# B&R Automation Studio project JOB_NUMBER (part 4)

```iecst
END_PROGRAM

PROGRAM _EXIT
  (* Insert code here *)
END_PROGRAM
```

### Device.typ
```iecst
TYPE
	Device_typ : 	STRUCT
		RequestRelease : UINT; (*The device wants to release, Will be a line destination OR DEVICE_RELEASE_ID if not destination in bag*)
		ReadyToRecieve : BOOL; (*The device is able to recieve a bag *)
		RecieveFromID : UINT; (*(Normally 0, But when using a point with multiple options set the ID we want to release)*)
		Recieved : BOOL; (*The device has recieved a bag, instruct previous device to copy data*)
		BagInTransit : BOOL; (*The incoming device has sent a bag.*)
		ClearDestination : BOOL; (*Set this to indicate to the incoming device to clear the bag destination on data transfer.*)
		Bag : UINT; (*The bag number where to incoming device must copy data to.*)
	END_STRUCT;
END_TYPE
```

### Library Logical/http_Lib/KanHttp (IEC)
Depends on: AsHttp

#### Constants.var - Exported constants
```iecst
VAR CONSTANT
	API_UNKNOWN : USINT := 0;
	API_MAINTENANCE_CONFIRM_REENTRY : USINT := 1;
	API_CONFIG_LOAD_NEW : USINT := 2;
	API_DISCHARGER_SUBMIT : USINT := 3;
	API_DATA_ENTRY_PARTLOAD : USINT := 4;
	API_ABB_MANUAL_CMD : USINT := 10;
	API_CUSTOM_BELT_CONFIG : USINT := 90;
	API_CUSTOM_RESET_SAFETY : USINT := 91;
	API_CUSTOM_VC_COMMAND : USINT := 92;
	API_ST_FUNCTIONS : USINT := 99;
END_VAR
```

#### FindAPI.st
```iecst
(* *Get API name from URI *)
FUNCTION FindAPI

	Start := LEN(ServiceName) + 2;// We must add the / character and 1 to place the cursor on the first Letter of the API name.
	Length := FIND(URI,'?');
	IF (Length = 0) THEN
		Length := LEN(URI)- LEN(ServiceName) + 1;;
	ELSE
		Length := Length - LEN(ServiceName) - 2;
	END_IF;

	apiName := 	MID(URI,Length,Start);

	IF (apiName = 'ConfirmBagReEntry') THEN FindAPI := API_MAINTENANCE_CONFIRM_REENTRY;
	ELSIF (apiName = 'Functions') THEN FindAPI := API_ST_FUNCTIONS;
	ELSIF (apiName = 'SendBeltLoadingConfig') THEN FindAPI := API_CUSTOM_BELT_CONFIG;
	ELSIF (apiName = 'ResetSafety') THEN FindAPI := API_CUSTOM_RESET_SAFETY;
	ELSIF (apiName = 'load-config') THEN FindAPI := API_CONFIG_LOAD_NEW;
	ELSIF (apiName = 'discharger-submit') THEN FindAPI := API_DISCHARGER_SUBMIT;
	ELSIF (apiName = 'abb-manual-control') THEN FindAPI := API_ABB_MANUAL_CMD;
	ELSIF (apiName = 'part-load') THEN FindAPI := API_DATA_ENTRY_PARTLOAD;
	ELSE FindAPI := API_UNKNOWN;
	END_IF;

END_FUNCTION
```

### Program Logical/http_Lib/httpServer (IEC) - *Listen for http requests

#### _getLoadingData.st
```iecst
ACTION _getLoadingData:

	prg	:= 0;
	cat := 0;
	cus := 0;
	dst := 0;
	error := 0;
	found := 0;
	//Set common parameters of the function.
	getParameterName.searchString := requestData;
	getParameterName.searchOffset := 0;
	getParameterName.searchEndProperty := STRING_DOLLAR;

	//Find the category
	getParameterName.searchPropertyName := '"category":';
	getParameterName.searchEndProperty := ',';
	getParameterName();
	IF getParameterName.status = ERR_OK THEN
		cat := DINT_TO_UDINT(atoi(ADR(getParameterName.outputValue)));
	ELSE
		error := 2;
	END_IF;

	//Find the customer
	getParameterName.searchPropertyName := '"customer":';
	getParameterName.searchEndProperty := ',';
	getParameterName();
	IF getParameterName.status = ERR_OK THEN
		cus := DINT_TO_UDINT(atoi(ADR(getParameterName.outputValue)));
	ELSE
		error := 2;
	END_IF;

	//Find the destination
	getParameterName.searchPropertyName := '"destination":';
	getParameterName.searchEndProperty := ',';
	getParameterName();
	IF getParameterName.status = ERR_OK THEN
		dst := DINT_TO_USINT(atoi(ADR(getParameterName.outputValue)));
	ELSE
		error := 4;
	END_IF;

	//Find the program
	getParameterName.searchPropertyName := '"program":';
	getParameterName.searchEndProperty := ',';
	getParameterName();
	IF getParameterName.status = ERR_OK THEN
		prg := DINT_TO_USINT(atoi(ADR(getParameterName.outputValue)));
		bag ACCESS ADR(Bag[212]);
		found := found + 1;
		bag.Cat := cat;
		bag.Prg := prg;
		bag.Cus := cus;
		bag.Dst := dst;
	ELSE
		error := 3;
	END_IF;

	sendResponse := (found > 0);
	errorResponse := (error > 0);

END_ACTION
```

#### _httpServer.st
```iecst
ACTION _httpServer:

	//Force the server to restart when then restart the PLC. Stops the server from crashing during PLC transfer
	IF (httpServer.status = ERR_FUB_ENABLE_FALSE) THEN
		httpServer.enable := 1;
	END_IF;
	//Error Handling -- Return the code 400 (Baf if there is a process error

	IF errorResponse THEN
		responseHeader.status := '400 Bad Request';
		sendResponse := 1;
	ELSIF ton_httpTimeOut.Q THEN
		responseHeader.status := '408 Request Timeout';
		responseData := 'Response Timeout';
		sendResponse := 1;
	ELSIF sendResponse THEN;
		responseHeader.status := '200 OK';
	END_IF;

	httpServer.enable := 1;
	httpServer.send := sendResponse; // Send Response on Rising edge.
	httpServer.abort := abortResponse;	//Send abort Response on Rising Edge

	IF (overRideData.responseDataLen > 0) THEN
		httpServer.responseDataLen := overRideData.responseDataLen;
	ELSE
		httpServer.responseDataLen := brsstrlen(ADR(responseData));
	END_IF;
	IF overRideData.responseHeader.contentType <> '' THEN
		responseHeader.contentType := overRideData.responseHeader.contentType;
	ELSE
		responseHeader.contentType := 'text/plain';
	END_IF;
	IF overRideData.responseHeader.status <> '' THEN
		responseHeader.status := overRideData.responseHeader.status;
	END_IF;

	responseHeader.contentLength := httpServer.responseDataLen;

	httpServer();

	IF (httpServer.phase = httpPHASE_RECEIVED) AND NOT sendResponse THEN
		recieved := 1;
	ELSE
		recieved := 0;
	END_IF;
	//Clear the overrides
	overRideData.responseDataLen 			:= 0;
	overRideData.responseHeader				:= BLANK_RESPONSE_HEADER;

	sendResponse := 0;
	abortResponse := 0;
	errorResponse := 0;

	//Request Timeout
	ton_httpTimeOut(IN:= (httpServer.phase = httpPHASE_RECEIVED),PT:= 500);//500
END_ACTION
```

### Program Logical/http_Lib/zzHttpDriver (IEC, version 3.00.4)

#### Main.st - Init, cyclic, exit code
```iecst
//V2.00.1- First Release of Version Control - Remove all unused code- Removed temp memory for recieve data as this helps when we get a "Invalid Character error"
//V2.00.2 -- ADD: New error handling if we do not recieve data when expected.
//V2.00.3 -- ADD: Add http reply code to the http data type so we don;t have to decode the string in the user tasks
//V3.00.1 -- CHANGE: TR 23/08/2019 - Convert the driver to a state machine
//V3.00.2 -- FIX: When writing to reports the status is being set as disabled causing repeated writes -- Comment out in HTTP_CLIENT_PROCESS_REQUEST and it works.. It makes no sense!!
//V3.00.3 -- FIX: Found solution to 3.02. The original state was being set to DISABLE so the proces step was exiting incorrectly.
//V3.00.4 -- FIX: Issue with certain errors getting stuck on the abort step.
PROGRAM _INIT
	//Use Static code now but change to config file later..
	HTTP_Config.Host := '10.8.4.220';
	HTTP_Config.Port := 0;
	httpComm ACCESS ADR(HTTP_Comm[0]);

	pUrl 							:= ADR(URL);
	pRequestHeader 					:= ADR(requestHeader);
	pResponseHeader 				:= ADR(responseHeader);
	pStatistics 					:= ADR(Statistics);
	pHost 							:= ADR(requestHeader.host);

	http_Client.pUri 				:= pUrl;
	http_Client.option 				:= httpOPTION_HTTP_11;
	http_Client.pHost 				:= pHost;
	http_Client.pRequestHeader 		:= pRequestHeader;
	http_Client.pResponseHeader 	:= pResponseHeader;
	http_Client.pStatistics 		:= pStatistics;

	//Configure RequestHeader
	requestHeader.protocol := DEFAULT_REQUEST_HEADER.protocol; //'HTTP/1.1';
	requestHeader.contentType := DEFAULT_REQUEST_HEADER.contentType;//'text/plain';
	requestHeader.connection := DEFAULT_REQUEST_HEADER.connection;//'close';
	requestHeader.keepAlive := DEFAULT_REQUEST_HEADER.keepAlive;//'max=100,timeout=5';

	sizeTempMem := 500000; //Allocate 500k of free memory
	TMP_alloc(sizeTempMem,ADR(pTempMem));

	ringBuffer[0] := 0;
	//Check for any requests that were being processed on shut down..
	FOR n := 1 TO HTTP_MAX_COMM DO
		IF HTTP_Comm[n].Status = HTTP_COMM_STATUS_IN_PROCESS THEN
			ringBuffer[0] := n;
		ELSIF HTTP_Comm[n].Status = HTTP_COMM_STATUS_IN_BUFFER THEN
			ringBuffer[n] := n;
		END_IF;
	END_FOR;
	_orderRing;
END_PROGRAM

PROGRAM _CYCLIC

	//Listen to requests and add to ring buffer.
	_ringBuffer;
	http_Client.send	:= 0;
	http_Client.abort	:= 0;

	CASE httpState OF

		HTTP_CLIENT_WAIT_FOR_COMMAND: // Order the ring buffer and wait for a new command to be processed.
			http_Client.enable := 0;
			retryCount := 0;
			httpComm ACCESS ADR(HTTP_Comm[0]);
			//Wait for next command from ring buffer
			IF(ringBuffer[0] = 0) AND (ringBuffer[1] > 0) THEN
				ringBuffer[0] := ringBuffer[1];
				httpComm ACCESS ADR(HTTP_Comm[ringBuffer[0]]);
				httpComm.Status := HTTP_COMM_STATUS_IN_PROCESS;
				ringBuffer[1] := 0;
			ELSIF (ringBuffer[0] > 0) THEN
				httpState := HTTP_CLIENT_PROCESS_REQUEST;
			END_IF;

		HTTP_CLIENT_PROCESS_REQUEST:
			http_Client.enable := 0;

			replyCode := 0;
			status := HTTP_COMM_STATUS_IN_PROCESS;
			lastError := '';

			httpComm ACCESS ADR(HTTP_Comm[ringBuffer[0]]);

			brsmemcpy(ADR(URL),ADR(BLANK_CHARACTER),SIZEOF(URL));
			brsmemcpy(ADR(URL),httpComm.Command.Cmd_URL.Adr,httpComm.Command.Cmd_URL.Size);
			responseHeader := emptyResponseHeader;

			//Check for any overwrite of the host or header
			IF httpComm.Overwrite.RequestHeader THEN
				requestHeader.protocol 		:= httpComm.Overwrite.RequestHeader_Data.protocol;
				requestHeader.contentType 	:= httpComm.Overwrite.RequestHeader_Data.contentType;
				requestHeader.connection 	:= httpComm.Overwrite.RequestHeader_Data.connection;
				requestHeader.keepAlive 	:= httpComm.Overwrite.RequestHeader_Data.keepAlive;
			ELSE
				requestHeader.protocol 		:= DEFAULT_REQUEST_HEADER.protocol; //'HTTP/1.1';
				requestHeader.contentType 	:= DEFAULT_REQUEST_HEADER.contentType;//'text/plain';
				requestHeader.connection 	:= DEFAULT_REQUEST_HEADER.connection;//'close';
				requestHeader.keepAlive 	:= DEFAULT_REQUEST_HEADER.keepAlive;//'max=100,timeout=5';
			END_IF;
			IF httpComm.Overwrite.Host THEN
				requestHeader.host := httpComm.Overwrite.Host_Config.Host;
				HTTP_Config.Port := httpComm.Overwrite.Host_Config.Port;
			ELSE
				requestHeader.host := HTTP_Config.Host;
				HTTP_Config.Port := 0;
			END_IF;

			requestHeader.contentLength 	:= httpComm.Command.Body_Data.Size;
			http_Client.hostPort 			:= HTTP_Config.Port;
			http_Client.method 				:= httpComm.Command.Method;
			http_Client.pRequestData 		:= httpComm.Command.Body_Data.Adr;
			http_Client.requestDataLen 		:= httpComm.Command.Body_Data.Size;

			IF (httpComm.Command.ResponseData.Adr > 0) AND (httpComm.Command.ResponseData.Size > 0) THEN
				http_Client.pResponseData 	:= httpComm.Command.ResponseData.Adr;
				http_Client.responseDataSize := httpComm.Command.ResponseData.Size;
			ELSE
				http_Client.pResponseData := pTempMem;
				http_Client.responseDataSize := sizeTempMem;
			END_IF;
			IF (http_Client.status = ERR_FUB_ENABLE_FALSE) THEN
				httpState := HTTP_CLIENT_PROCESS_ENABLE;
			END_IF;

		HTTP_CLIENT_PROCESS_ENABLE:
			http_Client.enable := 1;
			IF (http_Client.status = ERR_OK) THEN
				httpState := HTTP_CLIENT_PROCESS_SEND;
			END_IF;

		HTTP_CLIENT_PROCESS_SEND:
			http_Client.enable := 1;
			http_Client.send := 1;
			IF (http_Client.phase = httpPHASE_SENDING) THEN
				httpState := HTTP_CLIENT_PROCESS_WAIT_RESP;
			ELSIF (http_Client.status <> ERR_OK) AND (http_Client.status <> ERR_FUB_BUSY) THEN
				httpState := HTTP_CLIENT_ABORT;
			ELSIF (http_Client.phase = httpPHASE_RECEIVED) AND (http_Client.httpStatus > 0) THEN
				httpState := HTTP_CLIENT_PROCESS_RESPONSE;
			END_IF;

		HTTP_CLIENT_PROCESS_WAIT_RESP:
			http_Client.enable := 1;
			IF (http_Client.phase = httpPHASE_RECEIVED) THEN
				httpState := HTTP_CLIENT_PROCESS_RESPONSE;
			ELSIF (http_Client.status <> ERR_OK) AND (http_Client.status <> ERR_FUB_BUSY) THEN
				httpState := HTTP_CLIENT_ABORT;
			END_IF;

		HTTP_CLIENT_PROCESS_RESPONSE:
			http_Client.enable := 1;
			IF (http_Client.status = ERR_OK) THEN
				replyCode := http_Client.httpStatus;
				CASE http_Client.httpStatus OF
					200..207:
						IF (responseHeader.contentLength > 0) THEN
							IF (responseHeader.contentLength <= httpComm.Command.ResponseData.Size) THEN
								status := HTTP_COMM_STATUS_COMPLETE;
							ELSE
								status := HTTP_COMM_STATUS_ERROR;
								lastError := 'Response data area to small';
							END_IF;
						ELSIF ((httpComm.Command.Method = httpMETHOD_POST) OR (httpComm.Command.Method = httpMETHOD_PUT)) THEN
							status := HTTP_COMM_STATUS_COMPLETE;
						END_IF;
					300..307:
						//Implementation not done
						status := HTTP_COMM_STATUS_ERROR;
						lastError := responseHeader.status;
					400..426: //Errors
						status := HTTP_COMM_STATUS_ERROR;
						lastError := responseHeader.status;
					500..510://Server Errors
						status	:= HTTP_COMM_STATUS_ERROR;
						lastError 	:= responseHeader.status;
					ELSE
						httpState 	:= HTTP_CLIENT_ABORT;
				END_CASE;
			ELSIF (http_Client.status = httpERR_BUFFER_SIZE) THEN	// Response buffer is too small -- Abort and try again with temp memory area

			ELSIF (http_Client.status <> ERR_FUB_BUSY) THEN	//http client failure.
				itoa(http_Client.status,ADR(lastError));
				httpState := HTTP_CLIENT_ABORT;
			END_IF;

			IF (status <> HTTP_COMM_STATUS_IN_PROCESS) THEN
				httpState := HTTP_CLIENT_COMPLETE;
			END_IF;

		HTTP_CLIENT_COMPLETE:
			count := count + 1;
			http_Client.enable := 0;
			httpComm.Status := status;
			httpComm.LastError := lastError;
			httpComm.ReplyCode := replyCode;
			ringBuffer[0] := 0;
			httpState := HTTP_CLIENT_WAIT_FOR_COMMAND;

		HTTP_CLIENT_ABORT:
			http_Client.enable := 1;
			http_Client.abort := 1;
			IF (http_Client.phase = httpPHASE_WAITING) OR (http_Client.phase = httpPHASE_NOT_CONNECTED)  THEN
				IF (retryCount > 0) THEN
					httpState := HTTP_CLIENT_COMPLETE;
					status := HTTP_COMM_STATUS_ERROR;
				ELSE
					retryCount := 1;
					httpState := HTTP_CLIENT_PROCESS_REQUEST;
				END_IF;
			ELSIF (http_Client.phase = httpPHASE_RECEIVED) THEN //???
				IF (retryCount > 0) THEN
					httpState := HTTP_CLIENT_COMPLETE;
					status := HTTP_COMM_STATUS_ERROR;
				ELSE
					retryCount := 1;
					httpState := HTTP_CLIENT_PROCESS_REQUEST;
				END_IF;
			END_IF;

	END_CASE;

	http_Client();

END_PROGRAM
PROGRAM _EXIT
	WHILE (http_Client.status <> ERR_OK) DO
		http_Client.enable := 1;
		http_Client.abort := 1;
		http_Client();
	END_WHILE;

END_PROGRAM
```

### Bag.typ
```iecst
TYPE
	Bag_typ : 	STRUCT
		Prg : USINT; (*Program*)
		Dst : USINT; (*Destination - Only Supertrack*)
		Wgt : UINT; (*Weight*)
		Cnt : UINT; (*Count (Items)*)
		State : UINT; (*Maintenance State WAS UR1*)
		Bid : UDINT; (*Bag ID - Supertrack ID*)
		Cat : UDINT; (*Category*)
		Mis : UDINT; (*Batch ID - MIS Mis Server*)
		Cus : UDINT; (*Customer *)
		BagNo : UDINT; (*Actual Bag Number // Was UR2*)
		Timestamp : DATE_AND_TIME;
	END_STRUCT;
END_TYPE
```

### SystemConstants.var - *SYSTEM Constants
```iecst
VAR CONSTANT
	MAX_CAMERAS : USINT := 0; (** Number of B&R Barcode scanners*)
	MAX_CONTACTRON : USINT := 0;
	MAX_DRIVES : USINT := 1; (*Set to number of drives*)
	MAX_DUAL_CHANNELS : USINT := 10; (** Number of Estops*)
	MAX_FUSE_BANKS : USINT := 0;
	MAX_HOIST : USINT := 6;
	MAX_RAILS : UINT := 201; (**DO NOT USE -> USE RAIL_COUNT INSTEAD*)
	MAX_SAFE_ZONES : USINT := 6;
END_VAR
```

### Program Logical/Standard/ABB_EPL/ABB_Driver (IEC, version 4.00.2)

#### Main.st - Init, cyclic, exit code
```iecst
//V2.00.1 -- First stable release
//V2.00.2 -- Set brake control to be optional - This means changing when we encode the paramater structure.
//V2.00.3 -- Add new constant to set MAX_FREQUENCY
//V2.00.4 -- If the drive started not on remote it wouldn;t always go into config to start. ADD new mode for when module ok is false.
//V2.00.5 -- Add test mode for simulation
//V2.00.6 -- BUG FIX -- Minumum speed was being set to Max which stopped speed control
//V2.00.7 -- REMOVE -- Remove the old structure for settings via http
//V2.00.8 -- FIX -- Correct the scaling of MaxCurrent from settings - we now us 200 = 2A
//V3.00.1 -- CHANGE Combine Settings task into driver- Remove parameters from EPL write and move to SDO configuration function block
//V3.00.2 -- ADD Manual control mode via http!
//V3.00.3 -- Convert Manual Control to mappView.
//V4.00.1 -- Automatically get node number from PV structure.
//V4.00.2 -- Move Control word states into the program as the were not being copy when the task was moved causing errors.
//V4.00.3 -- Change halt mode of belts to we do a proper decel

PROGRAM _INIT
	FOR n := 1 TO MAX_DRIVES DO
		drive ACCESS ADR(ABB_EPL.Drives[n]);
		drive.Comm.State := ABB_CONFIG;
		drive.Config.currentParam := 1; //Reset starting parameter index
		drive.Config.Node := 0;
		drive.Config.EPL_Address := '';
		index := 0;
		init_state := 0;
	END_FOR;

	FOR n := 1 TO 8 DO
		visu_manual[n].ListBoxVisible := 0;
		visu_manual[n].TargetVelocity := ABB_MIN_VELOCITY;
		visu_manual[n].selectedIndex := 0;
	END_FOR;

	IF (MAX_DRIVES > 8) THEN
		max_manualControls := 8;
	ELSIF (MAX_DRIVES > 1) THEN
		max_manualControls := MAX_DRIVES;
	ELSE
		max_manualControls := 1;
	END_IF;
	xRun := FALSE;
END_PROGRAM

PROGRAM _CYCLIC

	IF EDGENEG(xRun) THEN
		FOR n := 1 TO MAX_DRIVES DO
			drive ACCESS ADR(ABB_EPL.Drives[n]);
			drive.Comm.State := ABB_INIT;
			drive.Config.currentParam := 1; //Reset starting parameter index
			drive.Config.Node := 0;
			drive.Config.EPL_Address := '';
			index := 0;
			init_state := 0;
		END_FOR;
	ELSIF NOT xRun THEN
		_getNodeInfo;
	ELSE

		_manual;  // mappView manual control.
		FOR x := 1 TO MAX_DRIVES DO
			IF (testDrive > 0) THEN
				n := testDrive;
			ELSE
				n := x;
			END_IF;

			drive 		ACCESS ADR(ABB_EPL.Drives[n]);
			settings	ACCESS ADR(gSettings.Drive[n]);

			//Control Word												Status Word
			//Bit 0		Switch On										Bit 0	Ready To Switch On
			//Bit 1		Enable Voltage									Bit 1	Switched On
			//Bit 2		Quick Stop										Bit 2	Operation Enabled
			//Bit 3		Enable Operation								Bit 3	Fault
			//Bit 4		Not Used In Scalor Mode							Bit 4	Voltage Enabled
			//Bit 5		Not Used In Scalor Mode							Bit 5	Quick Stop
			//Bit 6		Not Used In Scalor Mode							Bit 6	Switch On Disabled
			//Bit 7		Fault Reset										Bit 7 	Warning
			//Bit 8		Halt											Bit 8	Drive Specific TBC
			//Bit 9		Operation Mode Specific							Bit 9	Remote
			//Bit 10	Reserved	??Remote Control??					Bit 10	Target Reached
			//Bit 11	Drive Specific	TBC								Bit 11 	Internal Limit Reached
			//Bit 12	Drive Specific	TBC								Bit 12	Not Used In Scalor Mode
			//Bit 13	Drive Specific	TBC								Bit 13	Not Used In Scalor Mode
			//Bit 14	Drive Specific	TBC								Bit 14	Drive Specific TBC
			//Bit 15	Drive Specific	TBC								Bit 15	Drive Specific TBC

			//Use a local instance of controlword so we don't pass changing data to the drive while processing

			controlWord := SHUT_DOWN;	// 0000 0000 0111 0110

			//Encode the controlword and statusword
			_packData;

			IF Std.TestMode AND NOT drive.Comm.ModuleOk THEN // TEST MODE
				IF drive.Cmd.Run THEN
					drive.Comm.State := ABB_RUNNING;
				ELSE
					drive.Status.ReadyToRun := 1;
				END_IF;
			ELSIF NOT drive.Comm.ModuleOk THEN
				drive.Comm.State := ABB_DISCONNECTED;
			ELSIF (drive.Config.params[MAX_PARAMS].status <> 0) OR (drive.Config.currentParam < MAX_PARAMS) THEN
				drive.Comm.State := ABB_CONFIG;
			ELSIF NOT drive.Status.OnRemote THEN
				drive.Comm.State := ABB_OFF_REMOTE;
			ELSIF drive.Status.Tripped THEN
				drive.Comm.State := ABB_TRIPPED;
			ELSIF NOT drive.Cmd.QuickStop THEN	//Enable quick stop
				drive.Comm.State := ABB_QUICK_STOP;
			ELSIF drive.Status.SwitchOnInhibit THEN
				drive.Comm.State := ABB_SWITCH_ON_INHIBITED;
			ELSIF drive.Comm.ErrorCode = ABB_FAULT_STO THEN
				drive.Comm.State := ABB_STO;
			END_IF;

			CASE drive.Comm.State OF

				ABB_DISCONNECTED:
					drive.Config.currentParam := 1; // Force write of parameters

				ABB_CONFIG: //Wait for module OK to be TRUE
					_setParameters; //Write params
					IF drive.Comm.ModuleOk AND (drive.Config.params[MAX_PARAMS].status = 0) THEN
						drive.Comm.State := ABB_SWITCH_ON_INHIBITED;
					END_IF;

				ABB_SWITCH_ON_INHIBITED:	//Wait for quick stop and enable to be true
					IF NOT drive.Status.SwitchOnInhibit THEN
						drive.Comm.State := ABB_NOT_READY_TO_SWITCH_ON;
					END_IF;

				ABB_NOT_READY_TO_SWITCH_ON:
					IF drive.Status.ReadyToSwitchOn THEN
						drive.Comm.State := ABB_READY_TO_SWITCH_ON;
					END_IF;

				ABB_READY_TO_SWITCH_ON:
					controlWord := SWITCH_ON; //0000 0111 0111
					IF drive.Status.ReadyToRun THEN
						drive.Comm.State := ABB_READY_TO_RUN;
					END_IF;

				ABB_READY_TO_RUN:
					controlWord := SWITCH_ON; //0000 0111 0111
					IF drive.Cmd.Run AND (ABS(drive.Cmd.TargetVelocity) >= ABB_MIN_VELOCITY) AND NOT drive.Manual.Enable THEN //Check min frequency is met
						drive.Comm.State := ABB_RUNNING;
					ELSIF drive.Manual.Run AND (ABS(drive.Manual.Velocity) >= ABB_MIN_VELOCITY)  THEN
						drive.Comm.State := ABB_RUNNING;
					END_IF;

				ABB_RUNNING:
					controlWord := ENABLE_OPERATION; //0000 0111 1111
					IF NOT (drive.Cmd.Run AND NOT drive.Manual.Enable) AND NOT (drive.Manual.Run AND drive.Manual.Enable) THEN
						drive.Comm.State := ABB_RAMP_DOWN;
					END_IF;

				ABB_RAMP_DOWN:
					controlWord := RAMP_DOWN; //0001 0111 1111
					IF drive.Comm.StatusWord.11 = 0 AND drive.Comm.ActVelocity = 0 THEN
						drive.Comm.State := ABB_READY_TO_RUN;
					END_IF;

				ABB_QUICK_STOP:
					controlWord := QUICK_STOP; //0000 0111 0010
					IF drive.Comm.StatusWord.11 = 0 AND drive.Comm.ActVelocity = 0 AND drive.Cmd.QuickStop THEN
						drive.Comm.State := ABB_READY_TO_RUN;
					END_IF;

				ABB_TRIPPED: // AUTO Reseting -- We should change to manual reset..
					//We must wait for the drive to be ready for reset and give an edge.
						IF (drive.Comm.StatusWord.11 = 0) AND (drive.Comm.ActVelocity = 0) THEN
							IF settings.AutoReset THEN
								controlWord := FAULT_RESET;
							ELSIF drive.Manual.ErrorReset THEN
								controlWord := FAULT_RESET;
								drive.Manual.ErrorReset := FALSE; // Reset the command.
							ELSIF (drive.Comm.ErrorCode = 0) THEN
								controlWord := FAULT_RESET; // THE FAULT HAS BEEN CLEARED EXTERNALLY
							END_IF;
						ELSE
							controlWord := DISABLE_VOLTAGE; //0000 0000 0000
						END_IF;

					//We can auto reset here..but we should log an error somewhere..
					IF NOT drive.Status.Tripped THEN
						drive.Manual.ErrorReset := FALSE; // Reset the command.
						drive.Cmd.Reset	 		:= FALSE;
						drive.Comm.State := ABB_SWITCH_ON_INHIBITED;
					END_IF;

				ABB_OFF_REMOTE:
					//Remote control not active
					controlWord := SET_REMOTE;
					////				IF drive.Status.OnRemote THEN
					////					IF (drive.Config.params[MAX_PARAMS].status <> 0) THEN
					////						drive.Comm.State := ABB_CONFIG;
					////					ELSE
					////						drive.Comm.State := ABB_SWITCH_ON_INHIBITED;
					////					END_IF;
					////				END_IF;
					//				IF NOT Std.Drives_AllowLocalMode AND (drive.Config.params[13].data = Std.Drives_AllowLocalMode) THEN //Only reset the parameters if the local control mode has chnaged
					//					_encodeParameters;
					//					drive.Config.currentParam := 1; //Reset starting parameter index
					//				END_IF;
					//
				ABB_STO:
					IF drive.Comm.ErrorCode <> ABB_FAULT_STO THEN
						drive.Comm.State := ABB_SWITCH_ON_INHIBITED;
					END_IF;

			END_CASE;
			drive.Status.Running := (drive.Comm.State =  ABB_RUNNING);
			drive.Comm.ControlWord := controlWord;

			drive.Manual := DRIVE_MANUAL_DEFAULT;
		END_FOR;

	END_IF;

	//Temp code so that we can set a node number, The NODE must already be set to 1 (DEFAULT)
	IF (newNode > 0) THEN
		setNodeNumber.enable := 1;
		setNodeNumber.node := 1;
		setNodeNumber.index := 16#4033;
		setNodeNumber.subindex := 16#03;
		setNodeNumber.pData :=  ADR(newNode);
		setNodeNumber.datalen := 2;
		setNodeNumber();
		IF (setNodeNumber.status = ERR_OK) THEN
			newNode := 0;
		END_IF;
	ELSIF saveNewNode THEN
		saveVar := 1;
		setNodeNumber.enable := 1;
		setNodeNumber.node := 1;
		setNodeNumber.index := 16#4033;
		setNodeNumber.subindex := 16#1B;
		setNodeNumber.pData :=  ADR(saveVar);
		setNodeNumber.datalen := 2;
		setNodeNumber();
		IF (setNodeNumber.status = ERR_OK) THEN
			saveNewNode := 0;
		END_IF;
	ELSIF (factoryReset > 0) THEN
		saveVar := 34560;
		setNodeNumber.enable := 1;
		setNodeNumber.node := UINT_TO_USINT(factoryReset);
		setNodeNumber.index := 16#4060;
		setNodeNumber.subindex := 16#06;
		setNodeNumber.pData :=  ADR(saveVar);
		setNodeNumber.datalen := 2;
		setNodeNumber();
		IF (setNodeNumber.status = ERR_OK) THEN
			factoryReset := 0;
		END_IF;
	END_IF;

END_PROGRAM
```

#### setParameters.st
```iecst
ACTION _setParameters:

	CASE settings.MotorSize OF // Need to set these values correctly

		ABB_MOTOR_0_25KW:
			nominalCurrent_9906		:= 7; //0.68 A
			nominalPower_9910		:= 25; // 0.37 kW
			nominalSpeed_9909 		:= 1300;
			maxCurrent				:= 190;//1.9A

		ABB_MOTOR_0_37KW_0_91A_1374:
			nominalCurrent_9906		:= 9; //0.91 A
			nominalPower_9910		:= 37; // 0.37 kW
			nominalSpeed_9909 		:= 1374;
			maxCurrent 				:= 320; //3.2A

		ABB_MOTOR_0_37KW_0_97A_1342:
			nominalCurrent_9906		:= 10; //0.97 A
			nominalPower_9910		:= 37; // 0.37 kW
			nominalSpeed_9909 		:= 1342;
			maxCurrent 				:= 350; //3.5A

		ABB_MOTOR_0_37KW_1_14A_1380:
			nominalCurrent_9906		:= 7; //1.14 A
			nominalPower_9910		:= 37; // 0.37 kW
			nominalSpeed_9909 		:= 1380;
			maxCurrent 				:= 350;//3.5A

		ABB_MOTOR_0_75KW:
			nominalCurrent_9906		:= 18; //1.75 A
			nominalPower_9910		:= 75; // 0.75 kW
			nominalSpeed_9909 		:= 1440;
			maxCurrent 				:= 1170; //11.7A

		ABB_MOTOR_1_5KW:
			nominalCurrent_9906		:= 30;// 3 A?
			nominalPower_9910		:= 150;// 1.5kW
			nominalSpeed_9909 		:= 1450;
			maxCurrent 				:= 2200; //22A ???

		ABB_MOTOR_2_2KW_4_75A_1450:
			nominalCurrent_9906		:= 48; //4.75 A
			nominalPower_9910		:= 220; // 2.2 kW
			nominalSpeed_9909 		:= 1450;
			maxCurrent 				:= 3000; //30A ???

		ABB_MOTOR_3KW:
			nominalCurrent_9906		:= 64;
			nominalPower_9910		:= 300; // 3 kW
			nominalSpeed_9909 		:= 1456;
			maxCurrent 				:= 5248; //52.48

		ABB_MOTOR_CUSTOM: // Future  Alow Motor data to be set individaully
		//			nominalCurrent_9906		:= 0;
		//			nominalPower_9910		:= 0;
		//			nominalSpeed_9909 		:= 0;
		//			maxCurrent 				:= 0;

	END_CASE;

	accTime := REAL_TO_DINT(settings.AccTime * 1000);
	decTime := REAL_TO_DINT(settings.DecTime * 1000);

	//V2.00.2 Encode parameters
	_encodeParameters;

	drive.Config.function.enable := TRUE;																	//Enable function block

	IF (drive.Config.Node > 0) THEN
		drive.Config.function.node := drive.Config.Node; 														//Node number of drive, set in ABB_EPL[n].cmd.node if non standard.
		drive.Config.function.pDevice := ADR(drive.Config.EPL_Address);											//Set powerlink address in ABB_Driver init task
	ELSE
		//drive.Config.function.node := n + 100; //Set the default to drive + 100
	END_IF;
	IF (drive.Config.Node > 0) AND (drive.Config.currentParam <= MAX_PARAMS) THEN
		IF (drive.Config.params[drive.Config.currentParam].status > 0) THEN									//Call function only if not completed
			drive.Config.function.index := drive.Config.params[drive.Config.currentParam].index; 			//Powerlink index address
			drive.Config.function.subindex := drive.Config.params[drive.Config.currentParam].subIndex;		//Powerlink sub index address
			drive.Config.function.pData := ADR(drive.Config.params[drive.Config.currentParam].data);		//Value of data to write
			drive.Config.function.datalen := drive.Config.params[drive.Config.currentParam].datalen;		//Size of data type														//Call function
			IF (drive.Config.function.status = ERR_OK) THEN 												//Clear errors
				drive.Config.params[drive.Config.currentParam].status := 0;
				drive.Config.params[drive.Config.currentParam].errorInfo := 0;
				drive.Config.currentParam := drive.Config.currentParam + 1;
			ELSIF (drive.Config.function.status <> ERR_FUB_BUSY) AND (drive.Config.function.status <> ERR_FUB_ENABLE_FALSE) THEN //Store errors
				drive.Config.params[drive.Config.currentParam].status := drive.Config.function.status;
				drive.Config.params[drive.Config.currentParam].errorInfo := drive.Config.function.errorinfo;
				drive.Config.function.enable := FALSE;
				//			ELSIF drive.Config.function.status <> 20925 THEN;//ERR_PLMGR_STATION_NOT_ACTIVE THEN  //Only skip if the devuce is active																																					//Skip if other error to stop PLC hanging in bootup
				//				drive.Config.params[drive.Config.currentParam].status := drive.Config.function.status;
				//				drive.Config.params[drive.Config.currentParam].errorInfo := drive.Config.function.errorinfo;
				//				drive.Config.currentParam := drive.Config.currentParam + 1;
			END_IF;
			drive.Config.function();
		ELSE
			drive.Config.function.enable := FALSE;
		END_IF;
	END_IF;

	//Parameters should be loaded onto default settings.
	//to default the drive set 9606 t0 34560
	//Node ID (5103) has to be manually set

END_ACTION
```

### Hoist.typ - Local data types
```iecst
TYPE
	OpcUa_type : 	STRUCT
		VC : ARRAY[100..249]OF OpcUa_VC_type;
	END_STRUCT;
	OpcUa_VC_type : 	STRUCT
		Read : OpcUa_VC_Read_type;
		Write : OpcUa_VC_Write_type;
	END_STRUCT;
	OpcUa_VC_Write_type : 	STRUCT
		Heartbeat : BOOL;
		PermissionToMove : BOOL;
		TargetPosition : USINT;
		ReleaseBag : BOOL;
		ReceiveBag : BOOL;
		LoadBag : BOOL;
		BagInTransit : BOOL;
	END_STRUCT;
	OpcUa_VC_Read_type : 	STRUCT
		StatusInfo : STRING[80];
		ActPosition : REAL;
		PositionNo : USINT;
		ReleaseBag : BOOL;
		ReceiveBag : BOOL;
		Heartbeat : BOOL;
		ReadyToReceive : BOOL;
		Auto : BOOL;
		Manual : BOOL;
		Error : BOOL;
		Weight : DINT;
		IsHome : BOOL;
		BagOnCarriage : BOOL;
		ChuteBlocked : BOOL;
	END_STRUCT;
END_TYPE
```

### Program Logical/Standard/HoistLibrary/HoistServer (IEC)

#### Variables.var
```iecst
(****************************************************)
VAR
	MTBasicsPWM_0 : MTBasicsPWM;
	i : USINT;
	pHmiOpcUa : REFERENCE TO OpcUa_VC_type;
	selectedVC : UINT;
	pulse : MTBasicsPWM;
	hoist : REFERENCE TO OpcUa_VC_type;
	ton_simulateRecv : ARRAY[230..249] OF TON;
END_VAR
```

#### Main.st
```iecst
//V1.00.1  - TR - Add simulution mode.

PROGRAM _INIT

	selectedVC := 240;

END_PROGRAM

PROGRAM _CYCLIC

	MTBasicsPWM_0.DutyCycle		:= 50;
	MTBasicsPWM_0.Period		:= 2;
	MTBasicsPWM_0.Enable		:= TRUE;
	MTBasicsPWM_0(Enable:= TRUE,DutyCycle:= 50,Period:= 2,Update := 1);

	//FOR i := 38 TO 39 DO

pHmiOpcUa ACCESS ADR(OpcUa.VC[selectedVC]);

IF Std.TestMode THEN
		FOR i := 231 TO 249 DO

			hoist ACCESS ADR (OpcUa.VC[i]);

			hoist.Read.PositionNo 			:=	hoist.Write.TargetPosition;
			hoist.Read.Auto							:= 1;
			hoist.Read.ReadyToReceive 	:= 1;
			hoist.Read.IsHome						:= 1;

			ton_simulateRecv[i].IN 			:= 	hoist.Write.ReceiveBag;
			ton_simulateRecv[i].PT 			:= T#5s;
			ton_simulateRecv[i]();

			hoist.Read.ReceiveBag := ton_simulateRecv[i].Q;

			IF ton_simulateRecv[i].Q THEN
				hoist.Read.BagOnCarriage := 1;
			ELSIF hoist.Write.ReleaseBag THEN
				hoist.Read.BagOnCarriage := 0;
			END_IF;

		END_FOR;

ELSE
		FOR i := 231 TO 249 DO
			OpcUa.VC[i].Write.Heartbeat	:= MTBasicsPWM_0.Out; // NOT OpcUa.VC[i].Write.Heartbeat;
			//OpcUa.VC[i].Write.Heartbeat	:= pulse.Out;

			OpcUa.VC[i].Read.StatusInfo;
			OpcUa.VC[i].Read.ActPosition;
			OpcUa.VC[i].Read.PositionNo;
			OpcUa.VC[i].Read.ReceiveBag;
			OpcUa.VC[i].Read.ReleaseBag;
			OpcUa.VC[i].Read.Heartbeat;
			OpcUa.VC[i].Read.ReadyToReceive;

		END_FOR;

END_IF;

	(* Establish a connection to the client *)

(*	ReadHeartbeat;

	CASE Connect_to_OpcUaServer_step OF

		WAIT:

			IF Connect_OpcUa THEN

				Connect_to_OpcUaServer_step := CONNECT_TO_OPCUA;
			END_IF;

		CONNECT_TO_OPCUA:

			SessionConnectInfo_0.SecurityMsgMode := UASecurityMsgMode_None;
			SessionConnectInfo_0.SecurityPolicy := UASecurityPolicy_None;
			SessionConnectInfo_0.TransportProfile := UATP_UATcp;
			SessionConnectInfo_0.UserIdentityToken.UserIdentityTokenType := UAUITT_Anonymous;
			SessionConnectInfo_0.SessionTimeout := T#10m;
			SessionConnectInfo_0.MonitorConnection := T#10s;

			UA_Connect_0.ServerEndpointUrl := 'opc.tcp://10.44.10.244:4840';
			UA_Connect_0.Timeout := T#10s;
			UA_Connect_0.Execute := TRUE;
			UA_Connect_0.SessionConnectInfo := SessionConnectInfo_0;

			IF (UA_Connect_0.Done = 1) THEN
				UA_Connect_0.Execute := FALSE;
				Connect_OpcUa := FALSE;
				ConnectionHdl := UA_Connect_0.ConnectionHdl;
				Connect_to_OpcUaServer_step := GET_NAMESPACE;
			END_IF;

			IF (UA_Connect_0.Error = 1) THEN
				ConnectionHdl := 0;
				UA_Connect_0.Execute := FALSE;
				Connect_to_OpcUaServer_step := ERROR_OPCUA;
			END_IF;

		GET_NAMESPACE:

			UA_GetNamespaceIndex_0.ConnectionHdl := ConnectionHdl;
			UA_GetNamespaceIndex_0.NamespaceUri := 'urn:B&R/pv/';
			UA_GetNamespaceIndex_0.Timeout := T#5s;
			UA_GetNamespaceIndex_0.Execute := TRUE;

			IF (UA_GetNamespaceIndex_0.Done = 1) THEN
				NamespaceIndex := UA_GetNamespaceIndex_0.NamespaceIndex;
				UA_GetNamespaceIndex_0.Execute := FALSE;
				Connect_to_OpcUaServer_step := GET_NODE_HANDLE;
			END_IF;

			IF (UA_GetNamespaceIndex_0.Error = 1) THEN
				NamespaceIndex := 0;
				UA_GetNamespaceIndex_0.Execute := FALSE;
				Connect_to_OpcUaServer_step := ERROR_OPCUA;
			END_IF;

		GET_NODE_HANDLE:

			UANodeID_0[0].NamespaceIndex := NamespaceIndex;
			UANodeID_0[0].Identifier := '::Test_OpcUa_Client:WriteHeartbeat';
			UANodeID_0[0].IdentifierType := UAIdentifierType_String;

			UA_NodeGetHandleList_0.ConnectionHdl := ConnectionHdl;
			UA_NodeGetHandleList_0.NodeIDCount := 1;
			UA_NodeGetHandleList_0.NodeIDs := UANodeID_0;
			UA_NodeGetHandleList_0.Timeout := T#10s;
			UA_NodeGetHandleList_0.Execute := TRUE;

			IF (UA_NodeGetHandleList_0.Done = 1) THEN
				NodeHdls := UA_NodeGetHandleList_0.NodeHdls;
				UA_NodeGetHandleList_0.Execute := FALSE;
				Connect_to_OpcUaServer_step := READ_LIST;
			END_IF;

			IF (UA_NodeGetHandleList_0.Error = 1) THEN
				NodeHdls[0] := 0;

				UA_NodeGetHandleList_0.Execute := FALSE;
				Connect_to_OpcUaServer_step := ERROR_OPCUA;
			END_IF;

		READ_LIST:

			UANodeAdditionalInfo_0[0].AttributeId := UAAI_Value;
			UANodeAdditionalInfo_0[0].IndexRangeCount := 0;

			Variable_Rd0[0] := '::ServerTask:ReadHeartbeat';

			IF NOT UA_ReadList_0.Done THEN

				UA_ReadList_0
					(
					Execute := TRUE,
					ConnectionHdl := ConnectionHdl,
					NodeHdlCount := 1,
					NodeHdls := NodeHdls,
					NodeAddInfo := UANodeAdditionalInfo_0,
					Timeout := T#10s,
				Variables := Variable_Rd0);

				IF (UA_ReadList_0.Busy = 0) THEN
					UA_ReadList_0.Execute := FALSE;

					IF (UA_ReadList_0.Done = 1) THEN
						TimestampHeart := UA_ReadList_0.TimeStamps[0];

					END_IF;
					IF (UA_ReadList_0.Error = 1) THEN
						TimestampHeart := 0;
						Connect_to_OpcUaServer_step := ERROR_OPCUA;
					END_IF;
				END_IF;

			ELSIF StopReading THEN
				Connect_to_OpcUaServer_step := RELEASE_NODE;
				UA_ReadList_0.Execute := FALSE;

			ELSE
				UA_ReadList_0
					(
					Execute := FALSE,
					ConnectionHdl := ConnectionHdl,
					NodeHdlCount := 1,
					NodeHdls := NodeHdls,
					NodeAddInfo := UANodeAdditionalInfo_0,
					Timeout := T#10s,
				Variables := Variable_Rd0);
			END_IF;

		RELEASE_NODE:

			UA_NodeReleaseHandleList_0.ConnectionHdl := ConnectionHdl;
			UA_NodeReleaseHandleList_0.NodeHdlCount := 1;
			UA_NodeReleaseHandleList_0.NodeHdls := NodeHdls;
			UA_NodeReleaseHandleList_0.Timeout := T#10s;
			UA_NodeReleaseHandleList_0.Execute := TRUE;
			StopReading := FALSE;

			IF (UA_NodeReleaseHandleList_0.Done = 1) THEN
				NodeHdls[0] := 0;

				UA_NodeReleaseHandleList_0.Execute := FALSE;
				Connect_to_OpcUaServer_step := DISCONNECT_OPCUA;
			END_IF;

			IF (UA_NodeReleaseHandleList_0.Error = 1) THEN
				NodeHdls[0] := 0;

				UA_NodeReleaseHandleList_0.Execute := FALSE;
				Connect_to_OpcUaServer_step := ERROR_OPCUA;
			END_IF;

		DISCONNECT_OPCUA:

			UA_Disconnect_0.ConnectionHdl := ConnectionHdl;
			UA_Disconnect_0.Timeout := T#10s;
			UA_Disconnect_0.Execute := TRUE;

			IF (UA_Disconnect_0.Done = 1) THEN
				ConnectionHdl := 0;
				UA_Disconnect_0.Execute := FALSE;
				Connect_to_OpcUaServer_step := WAIT;
			END_IF;

			IF (UA_Disconnect_0.Error = 1) THEN
				ConnectionHdl := 0;
				UA_Disconnect_0.Execute := FALSE;
				Connect_to_OpcUaServer_step := ERROR_OPCUA;
			END_IF;

		ERROR_OPCUA:

	END_CASE;

	UA_Connect_0;
	UA_GetNamespaceIndex_0;
	UA_NodeGetHandleList_0;
	UA_NodeReleaseHandleList_0;
	UA_Disconnect_0;				*)

END_PROGRAM

PROGRAM _EXIT
	(* Insert code here *)

END_PROGRAM
```

### IOlink.typ
```iecst
TYPE
	contactron_visu_manual_typ : 	STRUCT
		Visible : BOOL; (**Are the controls Visible*)
		Name : STRING[50];
		Address : STRING[80]; (*Reference to the phyical location*)
		CommOk : BOOL;
		ActCurrent : DINT;
		ErrorCode : UINT;
		RunReverse : BOOL;
		RunForwards : BOOL;
		SetCurrent : INT;
		ErrorReset : BOOL;
		ErrorActive : BOOL;
		selectedIndex : UINT;
		selectedValue : STRING[10];
		refreshDropDown : R_TRIG;
		ListBoxVisible : BOOL;
		EnableRunReverse : BOOL;
		EnableRunForwards : BOOL;
		Enable : BOOL;
		Node : USINT;
	END_STRUCT;
	Contactron_Cmd_Type : 	STRUCT
		Reset_Manual : BOOL;
		Reset_Automatic : BOOL;
		Stop : BOOL;
		Run : BOOL;
		Direction : Contactron_Direction;
		Current : USINT; (*Sets the trip current, enable must be off to write*)
	END_STRUCT;
	Contactron_Comms_Type : 	STRUCT
		Write : Contactron_Outputs_Type;
		Read : Contactron_Inputs_Type;
	END_STRUCT;
	Contactron_Device_Type :
		(
		CONTACTRON_H5_3 := 0,
		CONTACTRON_H5_9 := 1,
		CONTACTRON_H3_3 := 2,
		CONTACTRON_H3_9 := 3
		);
	Contactron_Direction :
		(
		CONTACTRON_FORWARD := 0,
		CONTACTRON_REVERSE := 1
		);
	Contactron_Inputs_Type : 	STRUCT
		Diagnostics : USINT;
		CurrentStatus : USINT; (*Current trip level and trip status*)
		ThermalPercentOfMax : USINT;
		CurrentPercentOfMax : USINT;
		DeviceType : USINT; (*Type of contactron used*)
		CurrentActual : USINT; (*10mA*)
		Data : ARRAY[0..5]OF USINT;
	END_STRUCT;
	Contactron_Outputs_Type : 	STRUCT
		Control : USINT;
		NominalCurrent : USINT;
	END_STRUCT;
	Contactron_Status_Type : 	STRUCT
		Error : BOOL;
		STO_Active : BOOL;
		Device_Ok : BOOL;
		Overload_Warning : BOOL;
		MainsFailure : BOOL;
		PhaseLoss : BOOL;
		Current : REAL;
		DeviceType : Contactron_Device_Type;
	END_STRUCT;
	Contactron_Type : 	STRUCT  (*Parent structure to hold all Contactron structures*)
		Cmd : Contactron_Cmd_Type;
		Status : Contactron_Status_Type;
		Comms : Contactron_Comms_Type;
		Manual : contactron_visu_manual_typ;
	END_STRUCT;
	IO_Link_Type : 	STRUCT  (*Parent structure to hold all IO_Link device structures*)
		Contactron : ARRAY[0..MAX_CONTACTRON]OF Contactron_Type; (*Parent structure to hold all Contactron structures*)
	END_STRUCT;
END_TYPE

(**)
```

### Program Logical/Standard/IOLink/Contactron/Contactron (IEC, version 1.00.2)

#### Main.st - Init, cyclic, exit code
```iecst
(********************************************************************
 * COPYRIGHT --
 ********************************************************************
 * PROGRAM: IOLink
 * File: IOLink_Driver.s
 * Author: Stephen Healy NOT ANYMORE :)
 * Created: Sept 05, 2018
 ********************************************************************
 * Implementation OF PROGRAM IOLink
 ********************************************************************)
//V1.00.1 First Release
//V1.00.1 TR 10/11/2020  - Remove run signal from contactron when there is a fault to allow the error to be acknowledged.
//V1.00.2 TR 07/04/2021  - Add Test mode

PROGRAM _INIT

END_PROGRAM

PROGRAM _CYCLIC

	//Call contactron action
	IF MAX_CONTACTRON > 0 THEN
		_visu;
		_Contactron;

	END_IF;

END_PROGRAM
```

#### Variables.var - Local variables
```iecst
VAR
	n : UINT;
END_VAR
VAR CONSTANT
	max_manualControls : USINT := 8;
END_VAR
VAR
	visu_man : REFERENCE TO contactron_visu_manual_typ;
	visu_manual : ARRAY[0..max_manualControls] OF contactron_visu_manual_typ;
	selIndex : DINT;
	updateDropDown : BOOL;
	index : UINT;
	manualSelectDrowDown : ARRAY[0..MAX_CONTACTRON] OF STRING[125];
	sIndex : STRING[10];
	run : BOOL;
	contactron : REFERENCE TO Contactron_Type;
	RunMotor : BOOL;
	name : STRING[30];
END_VAR
VAR CONSTANT
	CONTACTRON_MANUAL_DEFAULT : contactron_visu_manual_typ := (RunReverse:=FALSE,RunForwards:=FALSE,ErrorReset:=FALSE,Enable:=FALSE);
END_VAR
```

#### _Contactron.st
```iecst
ACTION _Contactron:
	//----------------------------------------------
	//-----------------Contactron-------------------
	//----------------------------------------------

	//Write control word
	FOR n:=1 TO MAX_CONTACTRON DO
		contactron ACCESS ADR(IO_Link.Contactron[n]);

		IF Std.TestMode  THEN
			contactron.Status.Device_Ok := 1;
			IF contactron.Cmd.Run THEN
				contactron.Status.Current := 1.0;
			ELSE
				contactron.Status.Current := 0.0;
			END_IF;

		ELSE
			contactron.Comms.Read.CurrentActual 		:= contactron.Comms.Read.Data[0];
			contactron.Comms.Read.DeviceType 			:= contactron.Comms.Read.Data[1];
			contactron.Comms.Read.ThermalPercentOfMax 	:= contactron.Comms.Read.Data[2];
			contactron.Comms.Read.CurrentPercentOfMax 	:= contactron.Comms.Read.Data[3];
			contactron.Comms.Read.CurrentStatus 		:= contactron.Comms.Read.Data[4];
			contactron.Comms.Read.Diagnostics 			:= contactron.Comms.Read.Data[5];

			//Read status
			contactron.Status.Error 			:= contactron.Comms.Read.Diagnostics.0;
			contactron.Status.STO_Active 		:= NOT contactron.Comms.Read.Diagnostics.3;
			contactron.Status.Device_Ok 		:= contactron.Comms.Read.Diagnostics.5;
			contactron.Status.Overload_Warning 	:= contactron.Comms.Read.Diagnostics.6;
			contactron.Status.MainsFailure 		:= ((contactron.Comms.Read.CurrentStatus AND CONTACTRON_TRIP_STATUS) = CONTACTRON_MAINS_LOSS);
			contactron.Status.PhaseLoss 		:= ((contactron.Comms.Read.CurrentStatus AND CONTACTRON_TRIP_STATUS) = CONTACTRON_PHASE_LOSS);
			contactron.Status.Current 			:= contactron.Comms.Read.CurrentActual * 0.01;
			contactron.Status.DeviceType 		:= contactron.Comms.Read.DeviceType;

			IF contactron.Status.Error THEN
				run := 0;
//			ELSE IF contactron.Manaual.enable THEN
//				run := Manaul.run.
			ELSE
				run := contactron.Cmd.Run;
			END_IF;

			CASE contactron.Cmd.Direction OF
				CONTACTRON_FORWARD:
					contactron.Comms.Write.Control.0 := run;
					contactron.Comms.Write.Control.7 := run;
					contactron.Comms.Write.Control.1 := FALSE;
					contactron.Comms.Write.Control.5 := FALSE;

				CONTACTRON_REVERSE:
					contactron.Comms.Write.Control.0 := FALSE;
					contactron.Comms.Write.Control.7 := FALSE;
					contactron.Comms.Write.Control.1 := run;
					contactron.Comms.Write.Control.5 := run;

				ELSE
					contactron.Comms.Write.Control.0 := FALSE;
					contactron.Comms.Write.Control.7 := FALSE;
					contactron.Comms.Write.Control.1 := FALSE;
					contactron.Comms.Write.Control.5 := FALSE;

			END_CASE;

			contactron.Comms.Write.Control.2 := contactron.Cmd.Reset_Manual;
			contactron.Comms.Write.Control.3 := contactron.Cmd.Reset_Automatic;
			contactron.Comms.Write.Control.4 := FALSE; //NOT USED
			contactron.Comms.Write.Control.6 := contactron.Cmd.Stop;

			IF contactron.Cmd.Current > 0 THEN //Write trip current level
				contactron.Comms.Write.NominalCurrent := (contactron.Cmd.Current OR CONTACTRON_WRITE_CURRENT);
			ELSE
				contactron.Comms.Write.NominalCurrent := 0;
			END_IF;
			IF contactron.Cmd.Current = (contactron.Comms.Read.CurrentStatus AND CONTACTRON_CURRENT_STATUS) THEN
				contactron.Cmd.Current := 0; //Reset trip current if cmd written
			END_IF;

		END_IF;

		//Clear the manual commands.
		contactron.Manual := CONTACTRON_MANUAL_DEFAULT;
	END_FOR;
END_ACTION
```

#### _visu.st
```iecst
ACTION _visu:

	FOR n := 1 TO max_manualControls DO

		visu_man ACCESS ADR(visu_manual[n]);

		selIndex := atoi(ADR(visu_man.selectedValue));
		IF (selIndex > 0) AND (selIndex <= MAX_CONTACTRON) AND (selIndex <> visu_man.selectedIndex) THEN
			updateDropDown := 1;
			visu_man.selectedIndex := DINT_TO_UINT(selIndex);
		END_IF;

		visu_man.ListBoxVisible := (visu_man.selectedIndex = 0);

		visu_man.refreshDropDown.CLK := (visu_man.selectedIndex = 0);
		visu_man.refreshDropDown();
		IF visu_man.refreshDropDown.Q THEN
			updateDropDown := 1;
		END_IF;

		contactron ACCESS ADR(IO_Link.Contactron[visu_man.selectedIndex]);
		contactron.Manual.Enable := 1; //Mark Contactron as in manual mode

		visu_man.Visible 		:= (visu_man.selectedIndex >0);
		visu_man.Name    		:= gSettings.Contactron[visu_man.selectedIndex].Name;
//		visu_man.Node	 		:=
		visu_man.CommOk  		:= contactron.Status.Device_Ok;
		visu_man.ActCurrent 	:= contactron.Comms.Read.CurrentActual;
		visu_man.ErrorCode 		:= contactron.Status.Error;

		visu_man.ErrorActive := (contactron.Status.Error);

//		drive ACCESS ADR(ABB_EPL.Drives[visu_man.selectedIndex]);
//		drive.Manual.Enable 	:= 1; // Mark the drive as in manual mode.
//		drive.Manual.Velocity 	:= visu_man.TargetVelocity;
//
//		visu_man.Visible		:= (visu_man.selectedIndex > 0);
//		visu_man.Name			:= gSettings.Drive[visu_man.selectedIndex].Name;
//		visu_man.Node		 	:= drive.Config.Node;
//		visu_man.ModuleOk 		:= drive.Comm.ModuleOk;
//		visu_man.ActVelocity 	:= ABS(drive.Comm.ActVelocity);
//		visu_man.ActCurrent 	:= drive.Comm.ActCurrent;
//		visu_man.ActTorque 		:= drive.Comm.ActTorque;
//		visu_man.ErrorCode 		:= drive.Comm.ErrorCode;
//
//		visu_man.ErrorActive	:= (drive.Comm.State = ABB_TRIPPED);
//
		IF visu_man.ErrorReset THEN
			visu_man.ErrorReset := 0;
			contactron.Manual.ErrorReset := 1;
		END_IF;

//		CASE drive.Comm.State OF
//			ABB_INIT:
//				visu_man.State := '$$Drives.State.Init';
//			ABB_DISCONNECTED:
//				visu_man.State := '$$Drives.State.Disconnected';
//			ABB_QUICK_STOP:
//				visu_man.State := '$$Drives.State.QuickStop';
//			ABB_CONFIG:
//				visu_man.State := '$$Drives.State.Config';
//			ABB_SWITCH_ON_INHIBITED:
//				visu_man.State := '$$Drives.State.SwitchOnInhibit';
//			ABB_NOT_READY_TO_SWITCH_ON:
//				visu_man.State := '$$Drives.State.NotReady';
//			ABB_READY_TO_SWITCH_ON:
//				visu_man.State := '$$Drives.State.ReadyToSwitchOn';
//			ABB_READY_TO_RUN:
//				visu_man.State := '$$Drives.State.ReadyToRun';
//			ABB_RUNNING:
//				visu_man.State := '$$Drives.State.Running';
//			ABB_TRIPPED:
//				visu_man.State := '$$Drives.State.Tripped';
//			ABB_OFF_REMOTE:
//				visu_man.State := '$$Drives.State.OffRemote';
//			ABB_STO:
//				visu_man.State := '$$Drives.State.STO';
//			ABB_RAMP_DOWN:
//				visu_man.State := '$$Drives.State.RampDown';
//			ELSE
//				visu_man.State := '';
//		END_CASE;
//
		RunMotor := (contactron.Status.Device_Ok) AND NOT (contactron.Status.Error);
//		targetSpeedValid := ((visu_man.TargetVelocity >= ABB_MIN_VELOCITY) AND (visu_man.TargetVelocity <= ABB_MAX_VELOCITY) AND ((drive.Comm.State = ABB_READY_TO_RUN) OR  (drive.Comm.State = ABB_RUNNING)));
		//
		IF NOT visu_man.Enable THEN
			visu_man.RunReverse				:= 0;
			visu_man.RunForwards			:= 0;
			visu_man.EnableRunReverse   	:= 0;
			visu_man.EnableRunForwards		:= 0;
		ELSIF visu_man.RunForwards THEN
			contactron.Manual.RunForwards 	:= 1;
			contactron.Cmd.Run				:= RunMotor;
			visu_man.EnableRunReverse	  	:= 0;
		ELSIF visu_man.RunReverse THEN
			contactron.Manual.RunReverse	:= 1;
			contactron.Cmd.Run				:= RunMotor;
			visu_man.EnableRunForwards		:= 0;
		ELSE
			visu_man.EnableRunReverse		:= 1;
			visu_man.EnableRunForwards		:= 1;
		END_IF;

//		IF NOT targetSpeedValid THEN
//			visu_man.RunReverse 		:= 0;
//			visu_man.RunForwards 		:= 0;
//			visu_man.EnableRunReverse 	:= 0;
//			visu_man.EnableRunForwards 	:= 0;
//		ELSIF visu_man.RunForwards THEN
//			drive.Manual.Direction 	:= ABB_DIRECTION_FWD;
//			drive.Manual.Run		:= targetSpeedValid;
//			visu_man.EnableRunReverse := 0;
//		ELSIF visu_man.RunReverse THEN
//			drive.Manual.Direction 	:= ABB_DIRECTION_REV;
//			drive.Manual.Run		:= targetSpeedValid;
//			visu_man.EnableRunForwards := 0;
//		ELSE
//			visu_man.EnableRunReverse := 1;
//			visu_man.EnableRunForwards := 1;
//			drive.Manual.Run		:= 0;
//		END_IF;

	END_FOR;

	//Build the list box string;
	//[{'value':'text_1', 'text':'$$IAT/testText1'}, {'value':'text_2', 'text':'$$IAT/testText2'}]
	IF updateDropDown THEN
		index := 1;
		brsmemset(ADR(manualSelectDrowDown),0,SIZEOF(manualSelectDrowDown));
		manualSelectDrowDown[0] := '{"value":0,"text":""}';
		FOR n := 1 TO MAX_CONTACTRON DO
			contactron ACCESS ADR(IO_Link.Contactron[n]);
			IF NOT contactron.Manual.Enable THEN
				itoa(n,ADR(sIndex));

				IF (gSettings.Contactron[n].Name <> '') THEN
					name := gSettings.Contactron[n].Name;
				ELSE
					name := 'C ';
					brsstrcat(ADR(name),ADR(sIndex));
				END_IF;
				brsstrcat(ADR(manualSelectDrowDown[index]),ADR('{"value":"'));
				brsstrcat(ADR(manualSelectDrowDown[index]),ADR(sIndex));
				brsstrcat(ADR(manualSelectDrowDown[index]),ADR('","text":"'));
				brsstrcat(ADR(manualSelectDrowDown[index]),ADR(name));
				brsstrcat(ADR(manualSelectDrowDown[index]),ADR('"}'));
				index := index + 1;
			END_IF;
		END_FOR;
		updateDropDown := FALSE;
	END_IF;

END_ACTION
```

### Program Logical/Standard/IOLink/FuseManagement (IEC, version 1.00.2)

#### Main.st - Init, cyclic, exit code
```iecst
//V1.00.0 -- First Release
//V1.00.1 -- Update so we monitor the status of the fuse and can send reset commands
//V1.00.2 -- Invert the fault lamp to a healthy lamp to stay consistent with hardwired devices

PROGRAM _INIT
Fuse[1].pDevice := ADR('SL1.IF1.ST11.IF1.ST9.IF1');//'SL1.IF1.ST2.IF1.ST7.IF1');
Fuse[2].pDevice := ADR('SL1.IF1.ST11.IF1.ST9.IF2');
Fuse[3].pDevice := ADR('SL1.IF1.ST11.IF1.ST9.IF3');
Fuse[4].pDevice := ADR('SL1.IF1.ST11.IF1.ST9.IF4');
Fuse[5].pDevice := ADR('SL1.IF1.ST11.IF1.ST10.IF1');
Fuse[6].pDevice := ADR('SL1.IF1.ST11.IF1.ST10.IF2');
Fuse[7].pDevice := ADR('SL1.IF1.ST21.IF1.ST9.IF1');
Fuse[8].pDevice := ADR('SL1.IF1.ST21.IF1.ST9.IF2');
Fuse[9].pDevice := ADR('SL1.IF1.ST21.IF1.ST9.IF3');
Fuse[10].pDevice := ADR('SL1.IF1.ST21.IF1.ST9.IF4');
Fuse[11].pDevice := ADR('SL1.IF1.ST21.IF1.ST10.IF1');
Fuse[12].pDevice := ADR('SL1.IF1.ST21.IF1.ST10.IF2');
Fuse[13].pDevice := ADR('SL1.IF1.ST61.IF1.ST5.IF3');
Fuse[14].pDevice := ADR('SL1.IF1.ST61.IF1.ST5.IF4');
Fuse[15].pDevice := ADR('SL1.IF1.ST62.IF1.ST5.IF3');
Fuse[16].pDevice := ADR('SL1.IF1.ST62.IF1.ST5.IF4');
Fuse[17].pDevice := ADR('SL1.IF1.ST63.IF1.ST5.IF3');
Fuse[18].pDevice := ADR('SL1.IF1.ST63.IF1.ST5.IF4');

FOR n := 1 TO MAX_FUSE_BANKS DO
	fuse ACCESS ADR(Fuse[n]);
	fuse.Write.MinVoltage := 1500;
	fuse.Write.MaxVoltage := 2800;
	FOR i := 1 TO MAX_FUSES DO
      fuse.Write.Channel[i].Status := EB_STATE_ON;
      fuse.Write.Channel[i].TripCurrent := 40;
  END_FOR;
	fuse.index := 90;
	fuse.readStatusOnly := 0;
	fuseTrippedAlarm[n] := 0;
END_FOR;

//alarm 	ACCESS ADR(Alarm[208]);
END_PROGRAM

PROGRAM _CYCLIC

IF EDGEPOS(X[1003].X04) THEN
	reset[0] := 1;
END_IF;
IF EDGEPOS(X[2003].X04) THEN
	reset[1] := 1;
END_IF;

fuseFault[0] := 0;
fuseFault[1] := 0;
//alarm.On	:= 0;
//alarm.Name	:= 0;

FOR n := 1 TO MAX_FUSE_BANKS DO
	fuse ACCESS ADR(Fuse[n]);
	read ACCESS ADR(fuse.IOLinkRead);
	write ACCESS ADR(fuse.IOLinkWrite);

	read.enable := 1;
	write.enable := 1;
	write.pDeviceName 	:= fuse.pDevice;
	read.pDeviceName 	:= fuse.pDevice;

	IF EDGEPOS(read.readLen > 0) THEN
		count := count + 1;
	END_IF;

	IF (read.errorCode > 0) THEN
		fuse.index := 10;
	END_IF;

	IF (n < 5) THEN
		plc := 0;
	ELSE
		plc := 1;
	END_IF;

	CASE fuse.index	OF
		0:

		32:	//Read Error Count
			read.datatype 		:= ioLinkTYPE_SINT;
			read.pData			:= ADR(fuse.Read.ErrorCount);
			read.dataLen		:= SIZEOF(fuse.Read.ErrorCount);
			read.index			:= fuse.index;
			read.subIndex		:= 0;
			read();
			IF read.status = ERR_OK THEN
				fuse.index := fuse.index + 1;
			ELSIF (read.status <> ERR_FUB_BUSY) AND (read.status <> ERR_FUB_ENABLE_FALSE)  THEN
				fuse.index := fuse.index + 1;
				//fuse.Read.ErrorCount := 0;
			END_IF;

		33://
			fuse.index := 36;

		36://Device Status	 R/O USINT
			read.datatype 		:= ioLinkTYPE_SINT;
			read.pData			:= ADR(fuse.Read.DeviceStatus);
			read.dataLen		:= SIZEOF(fuse.Read.DeviceStatus);
			read.index			:= fuse.index;
			read.subIndex		:= 0;
			read();
			IF read.status = ERR_OK THEN
				fuse.index := fuse.index + 1;
			ELSIF (read.status <> ERR_FUB_BUSY) AND (read.status <> ERR_FUB_ENABLE_FALSE)  THEN
				fuse.index := fuse.index + 1;
				//fuse.Read.ErrorCount := 0;
			END_IF;

		37:// Device Status	 R/O String
			read.datatype 		:= ioLinkTYPE_STRING;
			read.pData			:= ADR(fuse.Read.DeviceStatusString);
			read.dataLen		:= SIZEOF(fuse.Read.DeviceStatusString);
			read.index			:= fuse.index;
			read.subIndex		:= 0;
			read();
			IF read.status = ERR_OK THEN
				fuse.index := fuse.index + 1;
			ELSIF (read.status <> ERR_FUB_BUSY) AND (read.status <> ERR_FUB_ENABLE_FALSE)  THEN
				fuse.index := fuse.index + 1;
				//fuse.Read.ErrorCount := 0;
			END_IF;

		38:
			fuse.index := 80;

		80://
			IF (fuse.trip > 0) THEN
				command := UINT_TO_USINT((fuse.trip * 5) - 2); // <--RESET //((fuse.trip * 5) - 4); //<-- ON

				write.datatype 		:= ioLinkTYPE_USINT;
				write.pData			:= ADR(command);
				write.dataLen		:= SIZEOF(command);
				write.index			:= fuse.index;
				write.subIndex		:= 0;
				write();
				IF (write.status = ERR_OK) THEN
					fuse.index := fuse.index + 1;	;
				ELSIF (write.status <> ERR_FUB_BUSY) AND (write.status <> ERR_FUB_ENABLE_FALSE) THEN
					fuse.index := fuse.index + 1;
				END_IF;
			ELSE
				fuse.index := fuse.index + 1;
			END_IF;

		81://Gateway options ? R/W
			IF fuse.Write.AutoNodeAllocation_Off OR fuse.Write.AutoNodeAllocation_On  THEN
				//1 is automatic allocation off!
				//0 is on?
				IF fuse.Write.AutoNodeAllocation_Off THEN
					write.datatype 		:= ioLinkTYPE_RECORD;
					gatewayOption 		:= 1;
					write.subIndex		:= 1;
				ELSE
					write.datatype 		:= ioLinkTYPE_SINT;
					gatewayOption 		:= 0;
					write.subIndex		:= 0 ;
				END_IF;
				write.pData			:= ADR(gatewayOption);
				write.dataLen		:= 1;
				write.index			:= fuse.index;
				write();
				IF (write.status = ERR_OK) THEN
					fuse.index := fuse.index + 1;	;
					fuse.Write.AutoNodeAllocation_On := 0;
					fuse.Write.AutoNodeAllocation_Off := 0;
				ELSIF (write.status <> ERR_FUB_BUSY) AND (write.status <> ERR_FUB_ENABLE_FALSE) THEN
					fuse.index := fuse.index + 1;
					fuse.Write.AutoNodeAllocation_On := 0;
					fuse.Write.AutoNodeAllocation_Off := 0;
				END_IF;

			ELSE // Read if no write
				read.datatype 		:= ioLinkTYPE_SINT;
				read.pData			:= ADR(fuse.Read.GatewayOptions);
				read.dataLen		:= SIZEOF(fuse.Read.GatewayOptions);
				read.index			:= fuse.index;
				read.subIndex		:= 0;
				read();
				IF read.status = ERR_OK THEN
					fuse.index := fuse.index + 1;
				ELSIF (read.status <> ERR_FUB_BUSY) AND (read.status <> ERR_FUB_ENABLE_FALSE)  THEN
					fuse.index := fuse.index + 1;
				END_IF;
			END_IF;

		82://Set breaker 1 options to all
			fuse.index := 90;

		83:// Reset individual breaker.

		90://Input Voltage
			read.datatype 		:= ioLinkTYPE_INT;
			read.pData			:= ADR(fuse.Read.InputVoltage);
			read.dataLen		:= SIZEOF(fuse.Read.InputVoltage);
			read.index			:= fuse.index;
			read.subIndex		:= 0;
			read();
			IF read.status = ERR_OK THEN
				fuse.index := fuse.index + 1;
			ELSIF (read.status <> ERR_FUB_BUSY) AND (read.status <> ERR_FUB_ENABLE_FALSE)  THEN
				fuse.index := fuse.index + 1;
			END_IF;

		91://Number of Nodes
			read.datatype 		:= ioLinkTYPE_USINT;
			read.pData			:= ADR(fuse.Read.NoNodes);
			read.dataLen		:= SIZEOF(fuse.Read.NoNodes);
			read.index			:= fuse.index;
			read.subIndex		:= 0;
			read();
			IF read.status = ERR_OK THEN
				IF (fuse.Read.NoNodes > MAX_FUSES) THEN
					fuse.Read.NoNodes := MAX_FUSES;
				END_IF;
				fuse.index := fuse.index + 1;
			ELSIF (read.status <> ERR_FUB_BUSY) AND (read.status <> ERR_FUB_ENABLE_FALSE)  THEN
				fuse.Read.NoNodes := 0;
				fuse.index := fuse.index + 1;
			END_IF;

		92://
			fuse.index := 100;

		100:// Max Voltage
			IF (fuse.Write.MaxVoltage > 0) THEN

				write.datatype 		:= ioLinkTYPE_INT;
				write.pData			:= ADR(fuse.Write.MaxVoltage);
				write.dataLen		:= SIZEOF(fuse.Write.MaxVoltage);
				write.index			:= fuse.index;
				write.subIndex		:= 0;
				write();
				IF (write.status = ERR_OK) THEN
					fuse.index := fuse.index + 1;
					fuse.Read.MaxVoltage := fuse.Write.MaxVoltage;
					fuse.Write.MaxVoltage := 0;
				ELSIF (write.status <> ERR_FUB_BUSY) AND (write.status <> ERR_FUB_ENABLE_FALSE) THEN
					fuse.index := fuse.index + 1;
					fuse.Write.MaxVoltage := 0;
				END_IF;
			ELSE // Read if no write

				read.datatype 		:= ioLinkTYPE_INT;
				read.pData			:= ADR(fuse.Read.MaxVoltage);
				read.dataLen		:= SIZEOF(fuse.Read.MaxVoltage);
				read.index			:= fuse.index;
				read.subIndex		:= 0;
				read();
				IF read.status = ERR_OK THEN
					fuse.index := fuse.index + 1;
				ELSIF (read.status <> ERR_FUB_BUSY) AND (read.status <> ERR_FUB_ENABLE_FALSE)  THEN
					fuse.index := fuse.index + 1;
					fuse.Read.MaxVoltage := 0;
				END_IF;
			END_IF;

		101://MinVoltage
			IF (fuse.Write.MinVoltage > 0) THEN
				write.datatype 		:= ioLinkTYPE_INT;
				write.pData			:= ADR(fuse.Write.MinVoltage);
				write.dataLen		:= SIZEOF(fuse.Write.MinVoltage);
				write.index			:= fuse.index;
				write.subIndex		:= 0;
				write();
				IF (write.status = ERR_OK) THEN
					fuse.index := fuse.index + 1;
					fuse.Read.MinVoltage :=	fuse.Write.MinVoltage;
					fuse.Write.MinVoltage := 0;
				ELSIF (write.status <> ERR_FUB_BUSY) AND (write.status <> ERR_FUB_ENABLE_FALSE) THEN
					fuse.index := fuse.index + 1;
					fuse.Write.MinVoltage := 0;
				END_IF;
			ELSE // Read if no write

				read.datatype 		:= ioLinkTYPE_INT;
				read.pData			:= ADR(fuse.Read.MinVoltage);
				read.dataLen		:= SIZEOF(fuse.Read.MinVoltage);
				read.index			:= fuse.index;
				read.subIndex		:= 0;
				read();
				IF read.status = ERR_OK THEN
					fuse.index := fuse.index + 1;
				ELSIF (read.status <> ERR_FUB_BUSY) AND (read.status <> ERR_FUB_ENABLE_FALSE)  THEN
					fuse.index := fuse.index + 1;
					fuse.Read.MinVoltage := 0;
				END_IF;
			END_IF;

		102:// Enable Events R/W
			IF (fuse.Write.EnableEvents > 0) THEN
				write.datatype 		:= ioLinkTYPE_SINT;
				write.pData			:= ADR(fuse.Write.EnableEvents);
				write.dataLen		:= SIZEOF(fuse.Write.EnableEvents);
				write.index			:= fuse.index;
				write.subIndex		:= 0;
				write();
				IF (write.status = ERR_OK) THEN
					fuse.index := fuse.index + 1;
					fuse.Write.EnableEvents := 0;
				ELSIF (write.status <> ERR_FUB_BUSY) AND (write.status <> ERR_FUB_ENABLE_FALSE) THEN
					fuse.index := fuse.index + 1;
					fuse.Write.EnableEvents := 0;
				END_IF;
			ELSE // Read if no write

				read.datatype 		:= ioLinkTYPE_SINT;
				read.pData			:= ADR(fuse.Read.EnableEvents);
				read.dataLen		:= SIZEOF(fuse.Read.EnableEvents);
				read.index			:= fuse.index;
				read.subIndex		:= 0;
				read();
				IF read.status = ERR_OK THEN
					fuse.index := fuse.index + 1;
				ELSIF (read.status <> ERR_FUB_BUSY) AND (read.status <> ERR_FUB_ENABLE_FALSE)  THEN
					fuse.index := fuse.index + 1;
					fuse.Read.EnableEvents := 0;
				END_IF;
			END_IF;

		103:
			fuse.index := 201;

		201..240://Read Only Trip Counter
			index := (fuse.index - 200);
			read.datatype 		:= ioLinkTYPE_SINT;
			read.pData			:= ADR(fuse.Read.Channel[index].TripCount);
			read.dataLen		:= SIZEOF(fuse.Read.Channel[index].TripCount);
			read.index			:= fuse.index;
			read.subIndex		:= 0;
			read();
			IF read.status = ERR_OK THEN
				fuse.index := fuse.index + 1;
			ELSIF (read.status <> ERR_FUB_BUSY) AND (read.status <> ERR_FUB_ENABLE_FALSE)  THEN
				fuse.index := fuse.index + 1;
				//fuse.Read.Channel[index].TripCount := 0;
			END_IF;

		241:
			fuse.index := 301;

		301..340://Read only Actaul Current
			index := (fuse.index - 300);
			read.datatype 		:= ioLinkTYPE_INT;
			read.pData			:= ADR(fuse.Read.Channel[index].ActCurrent);
			read.dataLen		:= SIZEOF(fuse.Read.Channel[index].ActCurrent);
			read.index			:= fuse.index;
			read.subIndex		:= 0;
			read();
			IF read.status = ERR_OK THEN
				IF (fuse.index < (300 + fuse.Read.NoNodes)) THEN
					fuse.index := fuse.index + 1;
				ELSE
					fuse.index := 401;
				END_IF;
			ELSIF (read.status <> ERR_FUB_BUSY) AND (read.status <> ERR_FUB_ENABLE_FALSE)  THEN
				IF (fuse.index < (300 + fuse.Read.NoNodes)) THEN
					fuse.index := fuse.index + 1;
				ELSE
					fuse.index := 401;
				END_IF;
			END_IF;

		341:
			fuse.index := 401;

		401..440://Over Current
			index := (fuse.index - 400);
			IF (fuse.Write.Channel[index].TripCurrent > 0) THEN
				write.datatype 		:= ioLinkTYPE_SINT;
				write.pData			:= ADR(fuse.Write.Channel[index].TripCurrent);
				write.dataLen		:= SIZEOF(fuse.Write.Channel[index].TripCurrent);
				write.index			:= fuse.index;
				write.subIndex		:= 0;
				write();
				IF (write.status = ERR_OK) THEN
					IF (fuse.index < (400 + fuse.Read.NoNodes)) THEN
						fuse.index := fuse.index + 1;
					ELSE
						fuse.index := 441;
					END_IF;
					fuse.Read.Channel[index].TripCurrent := fuse.Write.Channel[index].TripCurrent;
					fuse.Write.Channel[index].TripCurrent := 0;
				ELSIF (write.status <> ERR_FUB_BUSY) AND (write.status <> ERR_FUB_ENABLE_FALSE) THEN
					IF (fuse.index < (400 + fuse.Read.NoNodes)) THEN
						fuse.index := fuse.index + 1;
					ELSE
						fuse.index := 441;
					END_IF;
					fuse.Write.Channel[index].TripCurrent := 0;
				END_IF;
			ELSE // Read if no write

				read.datatype 		:= ioLinkTYPE_USINT;
				read.pData			:= ADR(fuse.Read.Channel[index].TripCurrent);
				read.dataLen		:= SIZEOF(fuse.Read.Channel[index].TripCurrent);
				read.index			:= fuse.index;
				read.subIndex		:= 0;
				read();
				IF read.status = ERR_OK THEN
					IF (fuse.index < (400 + fuse.Read.NoNodes)) THEN
						fuse.index := fuse.index + 1;
					ELSE
						fuse.index := 441;
					END_IF;
				ELSIF (read.status <> ERR_FUB_BUSY) AND (read.status <> ERR_FUB_ENABLE_FALSE)  THEN
					IF (fuse.index < (400 + fuse.Read.NoNodes)) THEN
						fuse.index := fuse.index + 1;
					ELSE
						fuse.index := 441;
					END_IF;
					fuse.Read.Channel[index].TripCurrent := 0;
				END_IF;
			END_IF;

		441..500:
			fuse.index := 501;
			fuse.trip := 0;

		501..540://	status RO
			index := (fuse.index - 500);

			read.datatype 		:= ioLinkTYPE_USINT;
			read.pData			:= ADR(fuse.Read.Channel[index].Status);
			read.dataLen		:= SIZEOF(fuse.Read.Channel[index].Status);
			read.index			:= fuse.index;
			read.subIndex		:= 0;
			read();
			IF read.status = ERR_OK THEN
				IF (fuse.index < (500 + fuse.Read.NoNodes)) THEN
					fuse.index := fuse.index + 1;
				ELSE
					fuse.index := 541;
				END_IF;
			ELSIF (read.status <> ERR_FUB_BUSY) AND (read.status <> ERR_FUB_ENABLE_FALSE)  THEN
				IF (fuse.index < (500 + fuse.Read.NoNodes)) THEN

					CASE fuse.Read.Channel[index].Status OF
						EB_STATE_NC:

						EB_STATE_OFF:

						EB_STATE_ON:

						EB_STATE_TRIP:
							fuse.trip := index;
						EB_STATE_I_90:

						EB_STATE_I_100:

						EB_STATE_TRIP_HARDWARE:

						EB_STATE_TRIP_THERMAL:
							fuse.trip := index;

						EB_STATE_TRIP_SW_OFF:

					END_CASE;

					fuse.index := fuse.index + 1;
				ELSE
					fuse.index := 541;
				END_IF;
				fuse.Read.Channel[index].Status := 0;
			END_IF;

		541:
			IF reset[plc] THEN
				fuse.index := 80;
			ELSIF fuse.readStatusOnly THEN
				fuse.index := 500;
			ELSE
				fuse.index := 901;
			END_IF;
			IF (fuse.trip > 0) THEN
				fuseTrippedAlarm[n] := 1;
			ELSE
				fuseTrippedAlarm[n] := 0;
			END_IF;

		701..740://Options

		901..940:
			index := (fuse.index - 900);
			read.datatype 		:= ioLinkTYPE_USINT;
			read.pData			:= ADR(fuse.Read.Channel[index].Type);
			read.dataLen		:= SIZEOF(fuse.Read.Channel[index].Type);
			read.index			:= fuse.index;
			read.subIndex		:= 0;
			read();
			IF read.status = ERR_OK THEN
				IF (fuse.index < (900 + fuse.Read.NoNodes)) THEN
					fuse.index := fuse.index + 1;
				ELSE
					fuse.index := 941;
				END_IF;
			ELSIF (read.status <> ERR_FUB_BUSY) AND (read.status <> ERR_FUB_ENABLE_FALSE)  THEN
				IF (fuse.index < (900 + fuse.Read.NoNodes)) THEN
					fuse.index := fuse.index + 1;
				ELSE
					fuse.index := 941;
				END_IF;
				//fuse.Read.Channel[index].ActCurrent := 0;
			END_IF;

		941:
			fuse.index := 501;
			fuse.readStatusOnly := 1;

		998:// Test Write
			write.pData := ADR(testData);
			write();
			IF (write.status = ERR_OK) THEN
				fuse.index := 1000;
			ELSIF (write.status <> ERR_FUB_BUSY) AND (write.status <> ERR_FUB_ENABLE_FALSE) THEN
				fuse.index := 1001;
			END_IF;
		999:// Test Read
			read();
			IF (read.status = ERR_OK) THEN
				fuse.index := 1000;
			ELSIF (read.status <> ERR_FUB_BUSY) AND (read.status <> ERR_FUB_ENABLE_FALSE)  THEN
				fuse.index := 1001;
			END_IF;
		1000:// Test result

	END_CASE;

	IF fuseTrippedAlarm[n] THEN
		fuseFault[plc]	:= 1;
		//alarm.On	:= TRUE;
		//alarm.Name	:= ALM_FUSE_TRIPPED;
	END_IF;

	IF NOT fuseFault[plc] THEN
		reset[plc] := 0;
	END_IF;

END_FOR;

Y[1004].Y02 := NOT fuseFault[0];
Y[2004].Y02 := NOT fuseFault[1];

END_PROGRAM
```

#### Variables.var - Local variables
```iecst
VAR
	lastIndex : UINT;
	fuseTrippedAlarm : ARRAY[0..MAX_FUSE_BANKS] OF BOOL; (*alarm : REFERENCE TO Alm;*)
	i : USINT;
	testData : INT;
	gatewayOption : BOOL;
	count : UDINT;
	command : USINT;
	reset : ARRAY[0..2] OF BOOL;
	fuseFault : ARRAY[0..2] OF BOOL;
	read : REFERENCE TO ioLinkRead;
	write : REFERENCE TO ioLinkWrite;
	fuse : REFERENCE TO Fuse_typ;
	n : INT;
	Fuse : ARRAY[0..MAX_FUSE_BANKS] OF Fuse_typ;
	index : UINT;
END_VAR
VAR CONSTANT
	MAX_FUSES : USINT := 40; (** Don;t set less than 40 the code will read the correct number*)
END_VAR
VAR
	plc : USINT;
END_VAR
```

#### Constants.var
```iecst
VAR CONSTANT
	EB_STATE_NC : USINT := 0; (*Not connected*)
	EB_STATE_OFF : USINT := 1; (*Switched Off*)
	EB_STATE_ON : USINT := 2; (*Switch On*)
	EB_STATE_TRIP : USINT := 3; (*Tripped*)
	EB_STATE_I_90 : USINT := 6; (*Current Exceeds 90%*)
	EB_STATE_I_100 : USINT := 14; (*Current Exceeds 100%*)
	EB_STATE_TRIP_HARDWARE : USINT := 18; (*Tripped - Hardware Error*)
	EB_STATE_TRIP_THERMAL : USINT := 20; (*Tripped - Thermal Release*)
	EB_STATE_TRIP_SW_OFF : USINT := 50; (*Switched Off*)
END_VAR
```

### Program Logical/Standard/IOLink/Fuses/FuseManagement

#### Main.st
```iecst
//V1.00.0 -- First Release
//V1.00.1 -- Update so we monitor the status of the fuse and can send reset commands
//V1.00.2 -- Invert the fault lamp to a healthy lamp to stay consistent with hardwired devices
//V1.00.3 -- 03 March 2021. Improve error handling, on IO link fault

//V2.00.1 -- 19/03/2021  - Rewrite for better performance and add mappview hooks
//V2.00.2	-- Refactor as io link has a limit of 7 simultaneous function blocks
//V2.00.3	-- Refactor as io link has a limit of 7 simultaneous function blocks  Read/Write combined. not exclusive
//V2.00.4 -- Add visualization code so we can read out the live values.
//V2.00.5 -- Add front end visu

PROGRAM _INIT
	Fuse[1].pDevice := ADR('SL1.IF1.ST2.IF1.ST8.IF1');
	Fuse[2].pDevice := ADR('SL1.IF1.ST2.IF1.ST8.IF2');
	Fuse[3].pDevice := ADR('SL1.IF1.ST2.IF1.ST8.IF3');
	Fuse[4].pDevice := ADR('SL1.IF1.ST2.IF1.ST8.IF4');
	Fuse[5].pDevice := ADR('SL1.IF1.ST3.IF1.ST2.IF1');
	//Fuse[6].pDevice := ADR('SL1.IF1.ST21.IF1.ST7.IF2');
	//Fuse[7].pDevice := ADR('SL1.IF1.ST21.IF1.ST7.IF3');
	//Fuse[8].pDevice := ADR('SL1.IF1.ST21.IF1.ST7.IF4');
	//
	//Fuse[9].pDevice := ADR('SL1.IF1.ST1.IF1.ST2.IF1');
	//Fuse[6].pDevice := ADR('SL1.IF1.ST21.IF1.ST10.IF2');
	//Fuse[7].pDevice := ADR('SL1.IF1.ST21.IF1.ST10.IF3');
	//Fuse[8].pDevice := ADR('SL1.IF1.ST21.IF1.ST10.IF4');

	gSettings.Fuse[1].GroupID := 'F71';
	gSettings.Fuse[2].GroupID := 'F72';
	gSettings.Fuse[3].GroupID := 'F73';
	gSettings.Fuse[4].GroupID := 'F81';
	gSettings.Fuse[5].GroupID := 'TTT';
	//Fuse[5].Settings.GroupID := 'F71';
	//Fuse[6].Settings.GroupID := 'F72';
	//Fuse[7].Settings.GroupID := 'F73';
	//Fuse[8].Settings.GroupID := 'F81';
	//Fuse[9].Settings.GroupID := 'TEST';
	//Fuse[7].Settings.GroupID := 'F77';
	//Fuse[8].Settings.GroupID := 'F78';

	visu_index := 1;
	//alarm 	ACCESS ADR(Alarm[208]);
	FOR n := 1 TO MAX_FUSE_BANKS DO
		visu_settings ACCESS ADR(gSettings.Fuse[n]);
		IF (visu_settings.MinVoltage = 0) THEN visu_settings.MinVoltage := 1900; END_IF;
		IF (visu_settings.MaxVoltage = 0) THEN visu_settings.MaxVoltage := 2850; END_IF;
		FOR i := 1 TO MAX_FUSE_CHANNELS DO
			IF (visu_settings.Channel[i].TripCurrent = 0) THEN visu_settings.Channel[i].TripCurrent := 40; END_IF;
			IF (visu_settings.Channel[i].FuseID = '') THEN
				brsitoa(i,ADR(sIndex));
				visu_settings.Channel[i].FuseID := Fuse[n].Settings.GroupID;
				brsstrcat(ADR(visu_settings.Channel[i].FuseID),ADR('.'));
				brsstrcat(ADR(visu_settings.Channel[i].FuseID),ADR(sIndex));
			END_IF;
		END_FOR;
	END_FOR;
END_PROGRAM

PROGRAM _CYCLIC

	IF EDGEPOS(X[1005].X04) THEN
		reset[0] := 1;
	END_IF;
	IF EDGEPOS(X[2005].X04) THEN
		reset[1] := 1;
	END_IF;

	fuseFault[0] := 0;
	fuseFault[1] := 0;
	//alarm.On	:= 0;
	//alarm.Name	:= 0;

	//	IF visu_id <= MAX_FUSE_BANKS THEN
	//	visu_data ACCESS ADR(Fuse[visu_id]);
	//ELSE
	//	visu_data ACCESS ADR(Fuse[0]);
	//END_IF;

	FOR n := 1 TO MAX_FUSE_BANKS DO
		fuse ACCESS ADR(Fuse[n]);

		fuse.Settings := gSettings.Fuse[n];

		//Set up and monitoring of the fuses
		_config;
		// Monitor the state for messaging and alarms.
		IF fuse.Info.NoNodes > 0 THEN
			FOR i := 1 TO fuse.Info.NoNodes DO
				CASE fuse.Info.Channel[i].Status OF
					EB_STATE_NC: // Not connected

					EB_STATE_OFF:

					EB_STATE_ON:

					EB_STATE_TRIP:
						fuseFault[1] := 1;

					EB_STATE_I_90:

					EB_STATE_I_100:

					EB_STATE_TRIP_HARDWARE: // Fuse failed

					EB_STATE_TRIP_THERMAL:
						fuseFault[1] := 1;

					EB_STATE_TRIP_SW_OFF: // Turned off by hand

				END_CASE;
			END_FOR;
		END_IF;

	END_FOR;

	// Read live values when required.
	_visuRead;

	//Y[1006].Y10 := NOT fuseFault[0];
	//Y[2006].Y10 := NOT fuseFault[1];

END_PROGRAM
```

### Modules.var
```iecst
VAR
	BusCouplerDiag : ARRAY[0..MAX_BUS_COUPLERS] OF BusCouplerDiag_typ;
END_VAR
VAR CONSTANT
	MAX_BUS_COUPLERS : UINT := 44;
END_VAR
```

### Package Logical/Standard/Settings - Looks after all PLC settings for drivers.

### Settings.typ
```iecst
TYPE
	settings_typ : 	STRUCT
		Camera : ARRAY[0..MAX_CAMERAS]OF Camera_Settings_typ;
		Drive : ARRAY[0..MAX_DRIVES]OF ABB_Settings_typ;
		Rail : ARRAY[0..MAX_RAILS]OF Rail_Permenant_typ;
		Fuse : ARRAY[0..MAX_FUSE_BANKS]OF FuseSetting_typ;
		Contactron : ARRAY[0..MAX_CONTACTRON]OF contactron_visu_manual_typ;
	END_STRUCT;
	Rail_Permenant_typ : 	STRUCT
		State : INT;
		Count : INT;
		RatchetPosition : INT;
	END_STRUCT;
END_TYPE
```

### Program Logical/Standard/Settings/Permenant (IEC, version 2.00.1) - *Store/Restore memory

#### Main.st - Init, cyclic, exit code
```iecst
PROGRAM _INIT
//Set all the rail states to perm.

FOR n := 1 TO MAX_RAILS DO
  //build the var_name;

  pSettings.Rail_Counter[n] := ADR(gSettings.Rail[n].Count);
  pSettings.Rail_State[n] := ADR(gSettings.Rail[n].State);
	pSettings.Rail_RatchetPosition[n] := ADR(gSettings.Rail[n].RatchetPosition);

  itoa(n,ADR(index_string));
  //r109.state
  var_name := 'r';
  brsstrcat(ADR(var_name),ADR(index_string));
  brsstrcat(ADR(var_name),ADR('.state'));
  // Get the Pointer address.
  IF (PV_xgetadr(ADR(var_name),ADR(pVar),ADR(sVar)) = 0) THEN
    p.Rail_State[n] := pVar;
    //brsmemcpy(p.Rail_State[n],pSettings.Rail_State[n],2);
  ELSE
    p.Rail_State[n] := 0;
  END_IF;

	var_name := 'r';
  brsstrcat(ADR(var_name),ADR(index_string));
  brsstrcat(ADR(var_name),ADR('.counter'));
  IF (PV_xgetadr(ADR(var_name),ADR(pVar),ADR(sVar)) = 0) THEN
    p.Rail_Counter[n] := pVar;
    //brsmemcpy(p.Rail_Counter[n],pSettings.Rail_Counter[n],2);
  ELSE
    p.Rail_Counter[n] := 0;
	END_IF;

	var_name := 'r';
	brsstrcat(ADR(var_name),ADR(index_string));
	brsstrcat(ADR(var_name),ADR('.ratchet_position'));
	IF (PV_xgetadr(ADR(var_name),ADR(pVar),ADR(sVar)) = 0) THEN
		p.Rail_RatchetPosition[n] := pVar;
		//brsmemcpy(p.Rail_Counter[n],pSettings.Rail_Counter[n],2);
	ELSE
		p.Rail_RatchetPosition[n] := 0;
	END_IF;

END_FOR;
init := TRUE;
END_PROGRAM

PROGRAM _CYCLIC
(*******************************
Update belt speeds.
*******************************)
// Set the values from eVue.

//beltSpeed[1] := Get_HigherByte(conveyor_module_1_value_1);
//beltSpeed[2] := Get_LowerByte(conveyor_module_1_value_1);
//beltSpeed[3] := Get_HigherByte(conveyor_module_1_value_2);
//beltSpeed[4] := Get_LowerByte(conveyor_module_1_value_2);
//beltSpeed[5] := Get_HigherByte(conveyor_module_1_value_3);
//beltSpeed[6] := Get_LowerByte(conveyor_module_1_value_3);

FOR n := 1 TO MAX_DRIVES DO
  IF (beltSpeed[n] > 0) AND (beltSpeed[n] <> gSettings.Drive[n].TargetVelocity) THEN
    gSettings.Drive[n].TargetVelocity := beltSpeed[n];
  ELSIF (gSettings.Drive[n].TargetVelocity = 0) THEN
    gSettings.Drive[n].TargetVelocity := ABB_MAX_VELOCITY;
  END_IF;
END_FOR;

FOR n := 1 TO MAX_RAILS DO
	IF init THEN
			IF (p.Rail_Counter[n] > 0) AND (pSettings.Rail_Counter[n] > 0) THEN
				brsmemcpy(p.Rail_Counter[n],pSettings.Rail_Counter[n],2);
			END_IF;
			IF (p.Rail_State[n] > 0) AND (pSettings.Rail_State[n] > 0) THEN
				brsmemcpy(p.Rail_State[n],pSettings.Rail_State[n],2);
			END_IF;
			IF (p.Rail_RatchetPosition[n] > 0) AND (pSettings.Rail_RatchetPosition[n] > 0) THEN
				brsmemcpy(p.Rail_RatchetPosition[n],pSettings.Rail_RatchetPosition[n],2);
			END_IF;
	ELSE
		IF (p.Rail_Counter[n] > 0) AND (pSettings.Rail_Counter[n] > 0) THEN
    	brsmemcpy(pSettings.Rail_Counter[n],p.Rail_Counter[n],2);
  	END_IF;
  	IF (p.Rail_State[n] > 0) AND (pSettings.Rail_State[n] > 0) THEN
    	brsmemcpy(pSettings.Rail_State[n],p.Rail_State[n],2);
		END_IF;
		IF (p.Rail_RatchetPosition[n] > 0) AND (pSettings.Rail_RatchetPosition[n] > 0) THEN
			brsmemcpy(pSettings.Rail_RatchetPosition[n],p.Rail_RatchetPosition[n],2);
		END_IF;
	END_IF;
END_FOR;

init := FALSE;

END_PROGRAM
```

#### Types.typ - Local data types
```iecst
TYPE
	Pointer_typ : 	STRUCT
		Rail_Counter : ARRAY[0..MAX_RAILS]OF UDINT;
		Rail_State : ARRAY[0..MAX_RAILS]OF UDINT;
		Rail_RatchetPosition : ARRAY[0..MAX_RAILS]OF UDINT;
	END_STRUCT;
END_TYPE
```

### Program Logical/Standard/Kanlink/zz_KanlinkConfig (IEC, version 1.20.0) - *Configuration of Kanlink

#### zz_KanlinkConfig.ab - Implementation code
```automation-basic
(********************************************************************
 * COPYRIGHT -- HP
 ********************************************************************
 * Program: zz_KanlinkConfig
 * File: zz_KanlinkConfig.ab
 * Author: treamsbottom
 * Created: September 07, 2012
 ********************************************************************
 * Implementation of program zz_KanlinkConfig
 ********************************************************************)
;Requirements
;From KGFramework
;	Libaries:
;		KgStdLib
;		KanLinkLib
;		mnParamLib
;	10ms Tasks:
;		hlKanLink
;	100ms Tasks:
;		svCPCache
;		mnEth
; When setting max connections for anything greater than 10
;the array decs will need changing. these are set by the constants HLKANLINK_MAX_CLIENTCONNS and HLKANLINK_MAX_SERVERCONNS in the frameworkshare
;Pkg_hlKanLink, KL_UserLib.Var
;----------------------------------------------------------------------------------------------------------------;
;-----21-1-2013..TR..Version A6 - First TestedVersion - Note Specials to run with Shuttle
;-----28-1-2013..TR..Version A7 - Remove Specials..Add option to send program and category number & Batch number.#
;-----03-03-2017..TR.Version A18 - Add "Advanced Connection Mode"
;-----07-06-2017 ..TR..Version A19 - Fix issues with sending empty bag date-- Remove reference to CAN[].Category -- Read all information from bag for consistency.
;-----------------------------------------------------------------------------------------------------------------
PROGRAM _INIT
	init := 0;
END_PROGRAM
PROGRAM _CYCLIC
;HLKANLINK_MAX_SERVERCONNS	;Declaration of max Server conns for KG Framework
;HLKANLINK_MAX_CLIENTCONNS	;Declaration of max Client conns for KG Framework
IF NOT init THEN
;Parameter Setup
;Global setting - Apply to all Kanlink Comms(Server,Client,OverView)
	Kanlink.GlobalSettings.TransferProgramCode 	= FALSE ; This transfers/Read the cat code to/from the bCustom area. Prg to/from sCategory
	Kanlink.GlobalSettings.TransferProgin_bCustom = FALSE ;This transfers/Read the Program code to/from the bCustom area. Category to/from sCategory
	Kanlink.GlobalSettings.UseBatchCode 		= TRUE	; Pass batch/SQL id
	Kanlink.GlobalSettings.BatchCodeTyp			= BatchTyp_UDINT  ;0 = UDINT, 1 = 16 byte unique (UDINT By default, extra code required for 16 byte )

;---------------------------------------------------------Batch Transfer Server---------------------------------------------------------------
;Server (Used to send data)		--------------------------- Variable = PT100
	Kanlink.Server.Enable = TRUE ; used to enable Server Comms
	Kanlink.Server.MaxConns	= 2 ; Number of Server connections
	 ; Start address of CAN variable
	;Address
	Kanlink.Server.IP[1].CommID = 1; //Opener 1
	Kanlink.Server.IP[1].Area 	= 3
	Kanlink.Server.IP[1].Adr 	= 11
;	Kanlink.Server.IP[1].AdvMode = FALSE // Use Advance mode- Pass in whole IP address as a string.
;	strcpy(ADR(Kanlink.Server.IP[1].AdrAdvMode),ADR("10.8.3.67"));
	Kanlink.Server.IP[1].CmdOpt = 0;

	Kanlink.Server.IP[2].CommID = 2; //Opener 2
	Kanlink.Server.IP[2].Area 	= 5
	Kanlink.Server.IP[2].Adr 	= 1
	Kanlink.Server.IP[2].CmdOpt = 0;

		;---------------------------------------------------------Batch transfer Client---------------------------------------------------------------
	;Client used to recieve data --------------------------- Variable = PTResp
	Kanlink.Client.Enable = TRUE ; used to enable Client Comms
	Kanlink.Client.MaxConns	= 1 ; Number of Client connections
	;Address

	Kanlink.Client.IP[1].CommID = 3	;//Transfer 1
	Kanlink.Client.IP[1].Area 	= 3
	Kanlink.Client.IP[1].Adr 	= 61
;	Kanlink.Client.IP[1].AdvMode = FALSE // Use Advance mode- Pass in whole IP address as a string.
;	strcpy(ADR(Kanlink.Client.IP[1].AdrAdvMode),ADR("10.8.4.20"));
	Kanlink.Client.IP[1].CmdOpt = 0

	Kanlink.Client.IP[1].CommID = 4	;//Transfer 2
	Kanlink.Client.IP[1].Area 	= 3
	Kanlink.Client.IP[1].Adr 	= 62
	;	Kanlink.Client.IP[1].AdvMode = FALSE // Use Advance mode- Pass in whole IP address as a string.
	;	strcpy(ADR(Kanlink.Client.IP[1].AdrAdvMode),ADR("10.8.4.20"));
	Kanlink.Client.IP[1].CmdOpt = 0
;

;

	//Sorting Rail
;	Kanlink.Client.IP[2].CommID = 4
;	Kanlink.Client.IP[2].Area 	= 3 ;Aero at sorting
;	Kanlink.Client.IP[2].Adr 	= 64
	;	Kanlink.Client.IP[1].AdvMode = FALSE // Use Advance mode- Pass in whole IP address as a string.
	;	strcpy(ADR(Kanlink.Client.IP[1].AdrAdvMode),ADR("10.8.4.20"));
;	Kanlink.Client.IP[2].CmdOpt = 1
;

;;---------------------------------------------------------Overview Server---------------------------------------------------------------
;	;------------------------------------------------Variable = STOverResp
;	;Use Overview Server.. SendData Data to Overview PLC - Only IP necessary - Client will request bag numbers.
	Kanlink.OverviewServer.Enable = FALSE
;	Kanlink.OverviewServer.MaxConns = 1
;
;	Kanlink.OverviewServer.IP[1].Area = 4
;	Kanlink.OverviewServer.IP[1].Adr = 21
;	Kanlink.OverviewServer.IP[1].AdvMode = FALSE
;	strcpy(ADR(Kanlink.OverviewServer.IP[1].AdrAdvMode),ADR("10.8.2.21"));
;
;	Kanlink.OverviewServer.IP[1].CmdOpt = 0
;;---------------------------------------------------------Overview Client---------------------------------------------------------------
;;------------------------------------------------Variable = STOverReq
;;Use Overview Client.. Recieve Data
	Kanlink.OverviewClient.Enable = FALSE
;	Kanlink.OverviewClient.MaxConns = 5
;	Kanlink.OverviewClient.CANOffset = 21
;;-----------PLC 1 - AERO SYSTEM
;	Kanlink.OverviewClient.StatusReg[1] = 951 ; D reg to map machine status for Tview.
;
;
;	Kanlink.OverviewClient.IP[1].Area = 3
;	Kanlink.OverviewClient.IP[1].Adr = 1	; To multiplex Edit KL_Overview
;	Kanlink.OverviewClient.IP[1].AdvMode = FALSE
;	strcpy(ADR(Kanlink.OverviewClient.IP[1].AdrAdvMode),ADR("10.8.3.1"));
;
;	Kanlink.OverviewClient.IP[1].CmdOpt = 0
;	//Batch data requested from Server
;	Kanlink.OverviewClient.InfoReq[1].wCntPositions = 6  ;Number of positions requested max 6 per request. If more than 6 set to 0 to multiplex...
;	Kanlink.OverviewClient.InfoReq[1].wNoOfPosition[0] = 1  ; Unqiue ID of data requested put all requests here if more than 6 the driver will multiplex the signals.
;	Kanlink.OverviewClient.InfoReq[1].wNoOfPosition[1] = 2	; There must be no gaps in the request numbers.	If not multiplexing, ensure index[6] = 0
;	Kanlink.OverviewClient.InfoReq[1].wNoOfPosition[2] = 3
;	Kanlink.OverviewClient.InfoReq[1].wNoOfPosition[3] = 4
;	Kanlink.OverviewClient.InfoReq[1].wNoOfPosition[4] = 5
;	Kanlink.OverviewClient.InfoReq[1].wNoOfPosition[5] = 6
;
;	//Bag number to map recieved data to.
;	Kanlink.OverviewClient.InfoResp[1].BagNum[0] = 501
;	Kanlink.OverviewClient.InfoResp[1].BagNum[1] = 502
;	Kanlink.OverviewClient.InfoResp[1].BagNum[2] = 503
;	Kanlink.OverviewClient.InfoResp[1].BagNum[3] = 504
;	Kanlink.OverviewClient.InfoResp[1].BagNum[4] = 505
;	Kanlink.OverviewClient.InfoResp[1].BagNum[5] = 506

;--------------------------------------------------------------END OF Configuration Code--------------------------------------------

;Check size of server and Client
	IF NOT Kanlink.Server.Enable THEN
		Kanlink.Server.MaxConns = 0
	ENDIF
	IF NOT Kanlink.Client.Enable THEN
		Kanlink.Client.MaxConns = 0
	ENDIF
	IF NOT Kanlink.OverviewServer.Enable THEN
		Kanlink.OverviewServer.MaxConns = 0
	ENDIF
	IF NOT Kanlink.OverviewClient.Enable THEN
		Kanlink.OverviewClient.MaxConns = 0
	ENDIF
	IF ((Kanlink.Server.MaxConns + Kanlink.OverviewServer.MaxConns) <= HLKANLINK_MAX_SERVERCONNS) THEN
		ServerDecOK = TRUE
	ELSE
		strcpy(ADR(Kanlink.ErrorString),"Declaration of HLKANLINK_MAX_SERVERCONNS not large enough")
		ServerDecOK = FALSE
	ENDIF
	IF ((Kanlink.Client.MaxConns + Kanlink.OverviewClient.MaxConns) <= HLKANLINK_MAX_CLIENTCONNS) THEN
		ClientDecOK = TRUE
	ELSE
		ClientDecOK = FALSE
		strcpy(ADR(Kanlink.ErrorString),"Declaration of HLKANLINK_MAX_CLIENTCONNS not large enough")
	ENDIF

	IF 	ServerDecOK AND ClientDecOK THEN

		;Server init
		IF Kanlink.Server.Enable THEN
			LOOP n = 1 TO Kanlink.Server.MaxConns DO
				;Build strings to pass to variable names, only required in a loop as index number changes.
				itoa(n,ADR(sn))	; put n into string
				strcpy(ADR(sReq),"PT100[");build string for variable name (request)
				strcat(ADR(sReq),ADR(sn))
				strcat(ADR(sReq),"].Req")
				strcpy(ADR(sResp),"PT100[");;build string for variable name (response)
				strcat(ADR(sResp),ADR(sn))
				strcat(ADR(sResp),"].Resp")
				IF Kanlink.Server.IP[n].AdvMode THEN
					IFhlKanLink.Parameter.Server[n].Adr = 0;
					IFhlKanLink.Parameter.Server[n].Area = 0
					IFhlKanLink.Parameter.Server[n].AdvMode := TRUE;
					strcpy(ADR(IFhlKanLink.Parameter.Server[n].AdrAdvMode),ADR(Kanlink.Server.IP[n].AdrAdvMode));
				ELSE
					IFhlKanLink.Parameter.Server[n].Adr = Kanlink.Server.IP[n].Adr ; Populate these arrays .
					IFhlKanLink.Parameter.Server[n].Area = Kanlink.Server.IP[n].Area
				ENDIF
				IFhlKanLink.Parameter.Server[n].Cmd = 1000 ; cmd from the server are always even
				IFhlKanLink.Parameter.Server[n].CmdOpt = Kanlink.Server.IP[n].CmdOpt
				IFhlKanLink.Parameter.Server[n].TimeOut = 1000 ;ms
				strcpy(ADR(IFhlKanLink.Parameter.Server[n].Name),"PT100") ; Diags Only
				strcpy(ADR(IFhlKanLink.Parameter.Server[n].sReq),ADR(sReq));"zzKanLink:PT100[0].Req")
				strcpy(ADR(IFhlKanLink.Parameter.Server[n].sResp),ADR(sResp));"zzKanLink:PT100[0].Resp")
			ENDLOOP
		ENDIF
		;Client Init
		IF Kanlink.Client.Enable THEN
			LOOP n = 1 TO Kanlink.Client.MaxConns DO
				itoa(n,ADR(sn))	; put n into string
				strcpy(ADR(sReq),"PTResp[");build string for variable name (request)
				strcat(ADR(sReq),ADR(sn))
				strcat(ADR(sReq),"].Req")
				strcpy(ADR(sResp),"PTResp[");;build string for variable name (response)
				strcat(ADR(sResp),ADR(sn))
				strcat(ADR(sResp),"].Resp")

				IF Kanlink.Client.IP[n].AdvMode THEN
					IFhlKanLink.Parameter.Client[n].Adr = 0;
					IFhlKanLink.Parameter.Client[n].Area = 0
					IFhlKanLink.Parameter.Client[n].AdvMode := TRUE;
					strcpy(ADR(IFhlKanLink.Parameter.Client[n].AdrAdvMode),ADR(Kanlink.Client.IP[n].AdrAdvMode));
				ELSE
					IFhlKanLink.Parameter.Client[n].Adr = Kanlink.Client.IP[n].Adr ; Populate these arrays .
					IFhlKanLink.Parameter.Client[n].Area = Kanlink.Client.IP[n].Area
				ENDIF
				IFhlKanLink.Parameter.Client[n].Cmd = 1000
				IFhlKanLink.Parameter.Client[n].CmdOpt = Kanlink.Client.IP[n].CmdOpt
				IFhlKanLink.Parameter.Client[n].CycleTime = 1000;ms
				strcpy(ADR(IFhlKanLink.Parameter.Client[n].Name),"PTResp")
				strcpy(ADR(IFhlKanLink.Parameter.Client[n].sReq),ADR(sReq))
				strcpy(ADR(IFhlKanLink.Parameter.Client[n].sResp),ADR(sResp))
			ENDLOOP
		ENDIF
		;Overview Server init
		;STOverResp[0] //Server sends batch data...
		IF Kanlink.OverviewServer.Enable THEN
			LOOP n = 1 TO Kanlink.OverviewServer.MaxConns DO
				;Build strings to pass to variable names, only required in a loop as index number changes.
				itoa(n,ADR(sn))	; put n into string
				strcpy(ADR(sReq),"STOverResp[");build string for variable name (request)
				strcat(ADR(sReq),ADR(sn))
				strcat(ADR(sReq),"].Req")
				strcpy(ADR(sResp),"STOverResp[");;build string for variable name (response)
				strcat(ADR(sResp),ADR(sn))
				strcat(ADR(sResp),"].Resp")

				Index = n + Kanlink.Server.MaxConns
				Kanlink.OverviewServer.IndexOffset = Kanlink.Server.MaxConns
				IF Kanlink.OverviewServer.IP[n].AdvMode THEN
					IFhlKanLink.Parameter.Server[Index].Adr = 0;
					IFhlKanLink.Parameter.Server[Index].Area = 0
					IFhlKanLink.Parameter.Server[Index].AdvMode := TRUE;
					strcpy(ADR(IFhlKanLink.Parameter.Server[Index].AdrAdvMode),ADR(Kanlink.OverviewServer.IP[n].AdrAdvMode));
				ELSE
					IFhlKanLink.Parameter.Server[Index].Adr = Kanlink.OverviewServer.IP[n].Adr ; Populate these arrays .
					IFhlKanLink.Parameter.Server[Index].Area = Kanlink.OverviewServer.IP[n].Area
				ENDIF

				IFhlKanLink.Parameter.Server[Index].Cmd = 1002 ;Batch Info Command
				IFhlKanLink.Parameter.Server[Index].CmdOpt = Kanlink.OverviewServer.IP[n].CmdOpt
				IFhlKanLink.Parameter.Server[Index].TimeOut = 1000 ;ms
				strcpy(ADR(IFhlKanLink.Parameter.Server[Index].Name),"STOverResp") ; Diags Only
				strcpy(ADR(IFhlKanLink.Parameter.Server[Index].sReq),ADR(sReq));"zzKanLink:STOverReq[0].Req")
				strcpy(ADR(IFhlKanLink.Parameter.Server[Index].sResp),ADR(sResp));"zzKanLink:STOverReq[0].Resp")

			ENDLOOP
		ENDIF

		;Kanlink OverView Client
		;STOverReq[0]// Client recieves batch data
		IF Kanlink.OverviewClient.Enable THEN
			LOOP n = 1 TO Kanlink.OverviewClient.MaxConns DO
				;Build strings to pass to variable names, only required in a loop as index number changes.
				itoa(n,ADR(sn))	; put n into string
				strcpy(ADR(sReq),"STOverReq[");build string for variable name (request)
				strcat(ADR(sReq),ADR(sn))
				strcat(ADR(sReq),"].Req")
				strcpy(ADR(sResp),"STOverReq[");;build string for variable name (response)
				strcat(ADR(sResp),ADR(sn))
				strcat(ADR(sResp),"].Resp")
				Index = n + Kanlink.Client.MaxConns
				Kanlink.OverviewClient.IndexOffset = Kanlink.Client.MaxConns

				IF Kanlink.OverviewClient.IP[n].AdvMode THEN
					IFhlKanLink.Parameter.Client[Index].Adr = 0;
					IFhlKanLink.Parameter.Client[Index].Area = 0
					IFhlKanLink.Parameter.Client[Index].AdvMode := TRUE;
					strcpy(ADR(IFhlKanLink.Parameter.Server[Index].AdrAdvMode),ADR(Kanlink.OverviewClient.IP[n].AdrAdvMode));
				ELSE
					IFhlKanLink.Parameter.Client[Index].Adr = Kanlink.OverviewClient.IP[n].Adr ; Populate these arrays .
					IFhlKanLink.Parameter.Client[Index].Area = Kanlink.OverviewClient.IP[n].Area
				ENDIF

				IFhlKanLink.Parameter.Client[Index].Cmd = 1002 ;Batch Info Command
				IFhlKanLink.Parameter.Client[Index].CmdOpt = Kanlink.OverviewClient.IP[n].CmdOpt
				IFhlKanLink.Parameter.Client[Index].CycleTime = 1000 ;ms
				strcpy(ADR(IFhlKanLink.Parameter.Client[Index].Name),"STOverReq") ; Diags Only
				strcpy(ADR(IFhlKanLink.Parameter.Client[Index].sReq),ADR(sReq));"zzKanLink:STOverResp[0].Req")
				strcpy(ADR(IFhlKanLink.Parameter.Client[Index].sResp),ADR(sResp));"zzKanLink:STOverResp[0].Resp")
			ENDLOOP
		ENDIF

		IFhlKanLink.in.xRestart = TRUE
		IFmnParam.Out.xParamOK = TRUE
		init = TRUE
		PT100 ; Variable that writes to the PT+ (Server)
		PTResp ; Variable that reads from PT+ (Client)
		STOverReq ;Variable used for the overview client
		STOverResp;Variable used for the overview server
	ENDIF//Server,client size OK
ENDIF//INIT

END_PROGRAM
```

### Program Logical/Standard/Kanlink/Kan_Driver (IEC) - *Kanlink Driver Server and Client
